# B&R Automation Studio project MotionTestBenchMaster (part 10)

#### Shift_Obj.st
```iecst
FUNCTION_BLOCK PhotoCell_SftObj
	IF IN_ConfigPresent THEN
		VAR_GrippersNumber	:= LIMIT(1, IN_GrippersNumber, CST_RepetitiveArrayDim);
		VAR_Mask 			:= IN_MaskEn AND HMI.Mask;

		IF VAR_Mask THEN
			VAR_Signal := IN_WaitOn AND NOT IN_WaitOff;
		ELSE
			VAR_Signal := IO.DI_Input;
		END_IF

		HMI.On := VAR_Signal;

		OUT	:= HMI.On;

		IF IN_MachinePitch AND IN_Enable THEN
			VAR_ActualValveCounter	:= INT_TO_USINT(FC_ReminderShift(VAR_ActualValveCounter	+ 1, VAR_GrippersNumber, 0));

			IF IN_WritePresenceEnable THEN //v1.63
				SHIFT_Position.ContainerPresence	:= IO.DI_Input;
			END_IF//v1.63

			IF SHIFT_Position.ContainerPresence THEN//v1.63
				IF NOT SHIFT_Position.ContainerBurst	AND	NOT VAR_Mask THEN//v1.63
					IF NOT IO.DI_Input THEN
						HMI.ConsecutiveErrors	:= SEL((IN_MStopConsecutiveValue > 0), 0,HMI.ConsecutiveErrors + 1);
						HMI.AbsoluteErrors		:= SEL((IN_CBlockAbsoluteValue > 0), 0, HMI.AbsoluteErrors + 1);
						HMI.TotalErrors			:= SEL((IN_MStopAbsoluteValue > 0), HMI.TotalErrors, HMI.TotalErrors + 1);

						VAR_RepetitiveCounterArray[VAR_ActualValveCounter]	:= SEL((IN_CBlockRepetitiveValue > 0), 0, VAR_RepetitiveCounterArray[VAR_ActualValveCounter] + 1);
						SHIFT_Position.ContainerPresence	:= FALSE;//v1.63

						IF VAR_RepetitiveCounterArray[VAR_ActualValveCounter] > IN_CBlockRepetitiveValue THEN
							OUT_CBlockRepetitive	:= TRUE;
						END_IF
					ELSE
						VAR_RepetitiveCounterArray[VAR_ActualValveCounter]	:= 0;
						HMI.ConsecutiveErrors	:= 0;//v1.63
					END_IF
				ELSE//v1.63
					VAR_RepetitiveCounterArray[VAR_ActualValveCounter]	:= 0;
					HMI.ConsecutiveErrors	:= 0;
				END_IF//v1.63
			END_IF

			HMI.AlwaysTrueSteps	:= SEL(VAR_EdgeChecked, HMI.AlwaysTrueSteps + 1, 0);//v1.63

			IF IN_CBlockRepetitiveValue > 0 THEN
				HMI.RepetitiveErrors	:= 0;

				FOR VAR_GrippersNumber:= 1	TO	CST_RepetitiveArrayDim	DO
					HMI.RepetitiveErrors := MAX(HMI.RepetitiveErrors, VAR_RepetitiveCounterArray[VAR_GrippersNumber]);
				END_FOR
			END_IF
		ELSIF NOT IO.DI_Input AND IN_Enable THEN
			VAR_EdgeChecked		:= TRUE;
		END_IF

		TMR_TON_TotalCounterReset(IN := IN_ResetCounters OR HMI.CounterReset, PT := T#5s);

		IF IN_ResetCounters OR HMI.CounterReset OR VAR_Mask OR NOT IN_Enable THEN
			IF NOT VAR_CounterResetMemory THEN
				VAR_CounterResetMemory	:= TRUE;

				FOR VAR_GrippersNumber:= 1 TO CST_RepetitiveArrayDim DO
					VAR_RepetitiveCounterArray[VAR_GrippersNumber]	:= 0;
					OUT_CBlockRepetitive	:= FALSE;
				END_FOR

				HMI.AlwaysTrueSteps		:= 0;
				HMI.RepetitiveErrors	:= 0;
				HMI.ConsecutiveErrors	:= 0;
				HMI.AbsoluteErrors		:= 0;
			END_IF
		ELSE
			VAR_CounterResetMemory	:= FALSE;
		END_IF

		IF TMR_TON_TotalCounterReset.Q THEN
			IF NOT VAR_TotalCounterResetMemory THEN
				VAR_TotalCounterResetMemory := TRUE;
				HMI.TotalErrors	:= 0;
			END_IF
		ELSE
			VAR_TotalCounterResetMemory := FALSE;
		END_IF

		HMI.ConfigPresent 	:= IN_ConfigPresent;
		HMI.ConfigAlarm 	:= IN_Alarm;
		HMI.Alarm 			:= OUT_CBlockAbsolute OR OUT_MStopConsecutive OR OUT_MStopAbsolute OR OUT_AlwaysTrueError;
		HMI.Wait			:= (IN_WaitOn AND NOT HMI.On) OR (IN_WaitOff AND HMI.On);
		HMI.MaskEnable		:= IN_MaskEn;

		OUT_CBlockAbsolute		:= (HMI.AbsoluteErrors 		>= IN_CBlockAbsoluteValue)		AND (IN_CBlockAbsoluteValue		> 0);
		OUT_MStopConsecutive	:= (HMI.ConsecutiveErrors 	>= IN_MStopConsecutiveValue)	AND (IN_MStopConsecutiveValue	> 0);
		OUT_MStopAbsolute		:= (HMI.AbsoluteErrors 		>= (IN_MStopAbsoluteValue + IN_CBlockAbsoluteValue))		AND (IN_MStopAbsoluteValue		> 0);	//V4.A.A.1.6.12
		OUT_AlwaysTrueError		:= (HMI.AlwaysTrueSteps		>= CST_AlwaysTrueMaxSteps)		AND (CST_AlwaysTrueMaxSteps		> 0);
	ELSE
		OUT						:= FALSE;
		OUT_CBlockRepetitive	:= FALSE;
		OUT_CBlockAbsolute		:= FALSE;
		OUT_MStopConsecutive	:= FALSE;
		OUT_MStopAbsolute		:= FALSE;
		OUT_AlwaysTrueError		:= FALSE;
		HMI.On 					:= FALSE;
		HMI.MaskEnable			:= FALSE;
		HMI.ConfigPresent 		:= FALSE;
		HMI.ConfigAlarm 		:= FALSE;
		HMI.Alarm 				:= FALSE;
		HMI.Wait				:= FALSE;
		HMI.RepetitiveErrors	:= 0;
		HMI.ConsecutiveErrors	:= 0;
		HMI.AbsoluteErrors		:= 0;
		HMI.AlwaysTrueSteps		:= 0;
	END_IF
END_FUNCTION_BLOCK

FUNCTION_BLOCK CapPhotoCell_SftObj
	IF IN_ConfigPresent THEN
		VAR_GrippersNumber	:= LIMIT(1, IN_GrippersNumber, CST_CounterArrayDim);
		VAR_Mask 			:= IN_MaskEn AND HMI.Mask;

		IF VAR_Mask THEN
			VAR_Signal := IN_WaitOn AND NOT IN_WaitOff;
		ELSE
			VAR_Signal := IO.DI_Input;
		END_IF

		HMI.On := VAR_Signal;

		OUT	:= HMI.On;

		IF IN_MachinePitch AND IN_Enable THEN
			VAR_ActualValveCounter	:= INT_TO_USINT(FC_ReminderShift(VAR_ActualValveCounter + 1, VAR_GrippersNumber, 0));

			IF SHIFT_Position.ContainerPresence AND SHIFT_Position.ClosingReleased AND NOT VAR_Mask THEN
				HMI.AlwaysTrueSteps	:= SEL(VAR_EdgeChecked, HMI.AlwaysTrueSteps + 1, 0);
				SHIFT_Position.ContainerClosed	:= IO.DI_Input;

				IF VAR_CapsReleased < 16#FFFFFFFF THEN
					VAR_CapsReleased := VAR_CapsReleased + 1;
				ELSE
					FOR VAR_i := VAR_AbsoluteErrorN TO 1 BY -1 DO
						VAR_AbsoluteCounterArray[VAR_i] := VAR_AbsoluteCounterArray[VAR_i] - (VAR_AbsoluteCounterArray[1] - 1);
					END_FOR
					VAR_CapsReleased := VAR_AbsoluteCounterArray[VAR_AbsoluteErrorN] + 1;
				END_IF

				IF NOT IO.DI_Input THEN
					HMI.ConsecutiveErrors	:= SEL((IN_MStopConsecutiveValue > 0), 0,HMI.ConsecutiveErrors + 1);
					//HMI.AbsoluteErrors		:= SEL((IN_CBlockAbsoluteValue > 0), 0, VAR_AbsoluteErrorN);	//V4.A.A.1.6.12
					HMI.TotalErrors			:= SEL((IN_CBlockAbsoluteValue > 0) OR (IN_MStopConsecutiveValue > 0), HMI.TotalErrors, HMI.TotalErrors + 1);

					VAR_RepetitiveCounterArray[VAR_ActualValveCounter] := SEL((IN_CBlockRepetitiveValue > 0), 0, VAR_RepetitiveCounterArray[VAR_ActualValveCounter] + 1);

					IF VAR_RepetitiveCounterArray[VAR_ActualValveCounter] > IN_CBlockRepetitiveValue THEN
						OUT_CBlockRepetitive	:= TRUE;
					END_IF

					IF IN_CBlockAbsoluteValue > 0 THEN
						IF IN_CBlockAbsoluteQuantity > 0 THEN
							VAR_AbsoluteCounterArray[VAR_AbsoluteErrorN] := VAR_CapsReleased;
						ELSE
							VAR_AbsoluteCounterArray[VAR_AbsoluteErrorN] := 0;
						END_IF

						VAR_AbsoluteErrorN := VAR_AbsoluteErrorN + 1;
					ELSE
						VAR_AbsoluteCounterArray[VAR_AbsoluteErrorN] := 0;
						VAR_AbsoluteErrorN := 1;
					END_IF
				ELSE
					VAR_RepetitiveCounterArray[VAR_ActualValveCounter]	:= 0;
					HMI.ConsecutiveErrors	:= 0; //v1.7.4
				END_IF
//			ELSE 								//v1.7.4
//				HMI.ConsecutiveErrors	:= 0;	//v1.7.4
			END_IF

			IF ((VAR_CapsReleased - VAR_AbsoluteCounterArray[1]) > IN_CBlockAbsoluteQuantity) AND (IN_CBlockAbsoluteQuantity > 0) THEN
				memmove(ADR(VAR_AbsoluteCounterArray[1]), ADR(VAR_AbsoluteCounterArray[2]), SIZEOF(VAR_AbsoluteCounterArray[1]) * 49);
				VAR_AbsoluteCounterArray[50] := 0;
				VAR_AbsoluteErrorN := MAX(VAR_AbsoluteErrorN - 1, 1);
			END_IF

			IF IN_CBlockRepetitiveValue > 0 THEN
				HMI.RepetitiveErrors := 0;
				FOR VAR_GrippersNumber:= 1 TO CST_CounterArrayDim DO
					HMI.RepetitiveErrors := MAX(HMI.RepetitiveErrors, VAR_RepetitiveCounterArray[VAR_GrippersNumber]);
				END_FOR
			END_IF

			HMI.AbsoluteErrors		:= SEL((IN_CBlockAbsoluteValue > 0), 0, VAR_AbsoluteErrorN - 1);	//V4.A.A.1.6.12
		ELSIF NOT IO.DI_Input AND IN_Enable THEN
			VAR_EdgeChecked := TRUE;
		ELSIF NOT IN_Enable THEN
			SHIFT_Position.ContainerClosed	:= SHIFT_Position.ContainerPresence AND SHIFT_Position.ClosingReleased;
		END_IF

		TMR_TON_TotalCounterReset(IN := IN_ResetCounters OR HMI.CounterReset, PT := T#5s);

		IF IN_ResetCounters OR HMI.CounterReset OR VAR_Mask OR NOT IN_Enable THEN
			IF NOT VAR_CounterResetMemory THEN
				VAR_CounterResetMemory	:= TRUE;

				FOR VAR_GrippersNumber:= 1 TO CST_CounterArrayDim DO
					VAR_RepetitiveCounterArray[VAR_GrippersNumber]	:= 0;
					OUT_CBlockRepetitive	:= FALSE;
				END_FOR

				memset(ADR(VAR_AbsoluteCounterArray[1]), 0, SIZEOF(VAR_AbsoluteCounterArray));
				VAR_AbsoluteErrorN := 1;

				VAR_CapsReleased		:= 0;
				HMI.AlwaysTrueSteps		:= 0;
				HMI.RepetitiveErrors	:= 0;
				//HMI.ConsecutiveErrors	:= 0;//V1.61
				HMI.AbsoluteErrors		:= 0;
			END_IF
		ELSE
			VAR_CounterResetMemory	:= FALSE;
		END_IF
		(*V1.61 Consecutive Errorors counter reset new management*)
		IF IN_ResetCountersConsecutive OR VAR_Mask OR NOT IN_Enable THEN
			IF NOT VAR_CounterConsResetMemory THEN
				VAR_CounterConsResetMemory	:= TRUE;
				HMI.ConsecutiveErrors	:= 0;
			END_IF
		ELSE
			VAR_CounterConsResetMemory	:= FALSE;
		END_IF

		IF TMR_TON_TotalCounterReset.Q THEN
			IF NOT VAR_TotalCounterResetMemory THEN
				VAR_TotalCounterResetMemory := TRUE;
				HMI.TotalErrors	:= 0;
			END_IF
		ELSE
			VAR_TotalCounterResetMemory := FALSE;
		END_IF

		HMI.ConfigPresent 	:= IN_ConfigPresent;
		HMI.ConfigAlarm 	:= IN_Alarm;
		HMI.Alarm 			:= OUT_CBlockAbsolute OR OUT_MStopConsecutive OR OUT_AlwaysTrueError;
		HMI.Wait			:= (IN_WaitOn AND NOT HMI.On) OR (IN_WaitOff AND HMI.On);
		HMI.MaskEnable		:= IN_MaskEn;

		OUT_CBlockAbsolute		:= (HMI.AbsoluteErrors 		>= IN_CBlockAbsoluteValue)		AND (IN_CBlockAbsoluteValue		> 0);
		OUT_MStopConsecutive	:= (HMI.ConsecutiveErrors 	>= IN_MStopConsecutiveValue)	AND (IN_MStopConsecutiveValue	> 0);
		OUT_AlwaysTrueError		:= (HMI.AlwaysTrueSteps		>= CST_AlwaysTrueMaxSteps)		AND (CST_AlwaysTrueMaxSteps		> 0);
	ELSE
		OUT						:= FALSE;
		OUT_CBlockRepetitive	:= FALSE;
		OUT_CBlockAbsolute		:= FALSE;
		OUT_MStopConsecutive	:= FALSE;
		OUT_AlwaysTrueError		:= FALSE;
		HMI.On 					:= FALSE;
		HMI.MaskEnable			:= FALSE;
		HMI.ConfigPresent 		:= FALSE;
		HMI.ConfigAlarm 		:= FALSE;
		HMI.Alarm 				:= FALSE;
		HMI.Wait				:= FALSE;
		HMI.RepetitiveErrors	:= 0;
		HMI.ConsecutiveErrors	:= 0;
		HMI.AbsoluteErrors		:= 0;
		HMI.AlwaysTrueSteps		:= 0;
	END_IF
END_FUNCTION_BLOCK

FUNCTION_BLOCK CapPhotoCell_SftObj_old
	IF IN_ConfigPresent THEN
		VAR_GrippersNumber	:= LIMIT(1, IN_GrippersNumber, CST_RepetitiveArrayDim);
		VAR_Mask 			:= IN_MaskEn AND HMI.Mask;

		IF VAR_Mask THEN
			VAR_Signal := IN_WaitOn AND NOT IN_WaitOff;
		ELSE
			VAR_Signal := IO.DI_Input;
		END_IF

		HMI.On := VAR_Signal;

		OUT	:= HMI.On;

		IF IN_MachinePitch AND IN_Enable THEN
			VAR_ActualValveCounter	:= INT_TO_USINT(FC_ReminderShift(VAR_ActualValveCounter + 1, VAR_GrippersNumber, 0));

			IF SHIFT_Position.ContainerPresence AND SHIFT_Position.ClosingReleased AND NOT VAR_Mask THEN
				HMI.AlwaysTrueSteps	:= SEL(VAR_EdgeChecked, HMI.AlwaysTrueSteps + 1, 0);
				SHIFT_Position.ContainerClosed	:= IO.DI_Input;

				IF NOT IO.DI_Input THEN
					HMI.ConsecutiveErrors	:= SEL((IN_MStopConsecutiveValue > 0), 0,HMI.ConsecutiveErrors + 1);
					HMI.AbsoluteErrors		:= SEL((IN_CBlockAbsoluteValue > 0), 0, HMI.AbsoluteErrors + 1);
					HMI.TotalErrors			:= SEL((IN_MStopAbsoluteValue > 0), HMI.TotalErrors, HMI.TotalErrors + 1);

					VAR_RepetitiveCounterArray[VAR_ActualValveCounter] := SEL((IN_CBlockRepetitiveValue > 0), 0, VAR_RepetitiveCounterArray[VAR_ActualValveCounter] + 1);

					IF VAR_RepetitiveCounterArray[VAR_ActualValveCounter] > IN_CBlockRepetitiveValue THEN
						OUT_CBlockRepetitive	:= TRUE;
					END_IF
				ELSE
					VAR_RepetitiveCounterArray[VAR_ActualValveCounter]	:= 0;
				END_IF
			ELSE
				HMI.ConsecutiveErrors	:= 0;
			END_IF

			IF IN_CBlockRepetitiveValue > 0 THEN
				HMI.RepetitiveErrors := 0;
				FOR VAR_GrippersNumber:= 1 TO CST_RepetitiveArrayDim DO
					HMI.RepetitiveErrors := MAX(HMI.RepetitiveErrors, VAR_RepetitiveCounterArray[VAR_GrippersNumber]);
				END_FOR
			END_IF
		ELSIF NOT IO.DI_Input AND IN_Enable THEN
			VAR_EdgeChecked := TRUE;
		ELSIF NOT IN_Enable THEN
			SHIFT_Position.ContainerClosed	:= SHIFT_Position.ContainerPresence AND SHIFT_Position.ClosingReleased;
		END_IF

		TMR_TON_TotalCounterReset(IN := IN_ResetCounters OR HMI.CounterReset, PT := T#5s);

		IF IN_ResetCounters OR HMI.CounterReset OR VAR_Mask THEN
			IF NOT VAR_CounterResetMemory THEN
				VAR_CounterResetMemory	:= TRUE;

				FOR VAR_GrippersNumber:= 1 TO CST_RepetitiveArrayDim DO
					VAR_RepetitiveCounterArray[VAR_GrippersNumber]	:= 0;
					OUT_CBlockRepetitive	:= FALSE;
				END_FOR

				HMI.AlwaysTrueSteps		:= 0;
				HMI.RepetitiveErrors	:= 0;
				HMI.ConsecutiveErrors	:= 0;
				HMI.AbsoluteErrors		:= 0;
			END_IF
		ELSE
			VAR_CounterResetMemory	:= FALSE;
		END_IF

		IF TMR_TON_TotalCounterReset.Q THEN
			IF NOT VAR_TotalCounterResetMemory THEN
				VAR_TotalCounterResetMemory := TRUE;
				HMI.TotalErrors	:= 0;
			END_IF
		ELSE
			VAR_TotalCounterResetMemory := FALSE;
		END_IF

		HMI.ConfigPresent 	:= IN_ConfigPresent;
		HMI.ConfigAlarm 	:= IN_Alarm;
		HMI.Alarm 			:= OUT_CBlockAbsolute OR OUT_MStopConsecutive OR OUT_MStopAbsolute OR OUT_AlwaysTrueError;
		HMI.Wait			:= (IN_WaitOn AND NOT HMI.On) OR (IN_WaitOff AND HMI.On);
		HMI.MaskEnable		:= IN_MaskEn;

		OUT_CBlockAbsolute		:= (HMI.AbsoluteErrors 		>= IN_CBlockAbsoluteValue)		AND (IN_CBlockAbsoluteValue		> 0);
		OUT_MStopConsecutive	:= (HMI.ConsecutiveErrors 	>= IN_MStopConsecutiveValue)	AND (IN_MStopConsecutiveValue	> 0);
		OUT_MStopAbsolute		:= (HMI.AbsoluteErrors 		>= IN_MStopAbsoluteValue)		AND (IN_MStopAbsoluteValue		> 0);
		OUT_AlwaysTrueError		:= (HMI.AlwaysTrueSteps		>= CST_AlwaysTrueMaxSteps)		AND (CST_AlwaysTrueMaxSteps		> 0);
	ELSE
		OUT						:= FALSE;
		OUT_CBlockRepetitive	:= FALSE;
		OUT_CBlockAbsolute		:= FALSE;
		OUT_MStopConsecutive	:= FALSE;
		OUT_MStopAbsolute		:= FALSE;
		OUT_AlwaysTrueError		:= FALSE;
		HMI.On 					:= FALSE;
		HMI.MaskEnable			:= FALSE;
		HMI.ConfigPresent 		:= FALSE;
		HMI.ConfigAlarm 		:= FALSE;
		HMI.Alarm 				:= FALSE;
		HMI.Wait				:= FALSE;
		HMI.RepetitiveErrors	:= 0;
		HMI.ConsecutiveErrors	:= 0;
		HMI.AbsoluteErrors		:= 0;
		HMI.AlwaysTrueSteps		:= 0;
	END_IF
END_FUNCTION_BLOCK

FUNCTION_BLOCK Ejector_SftObj
	VAR_Mask	:= HMI.Mask AND IN_MaskEn;

	(* Local *)
	IF IN_ManEn AND NOT IN_HMIAutoForce THEN
		VAR_ManOn	:= HMI.ManOn;
		VAR_Auto	:= NOT HMI.ManOff AND NOT HMI.ManOn;
	ELSE
		VAR_ManOn	:= FALSE;
		VAR_Auto	:= TRUE;
		HMI.ManOn	:= FALSE;
		HMI.ManOff	:= FALSE;
	END_IF

	IF IN_MachinePitch THEN
		VAR_AutoCnd := IN_ShiftPosition.ContainerPresence		AND (IN_ShiftPosition.ContainerBurst	OR
						(NOT IN_ShiftPosition.ContainerFilled	AND IN_FillingErrorEject) OR IN_ShiftPosition.EjectContainer) AND NOT VAR_Mask; (*V1.61*)
		IF VAR_AutoCnd AND NOT IN_SamplingModeActive THEN (*V1.61*)
			HMI.ConsecutiveErrors	:= HMI.ConsecutiveErrors	+ 1;
			HMI.AbsoluteErrors		:= HMI.AbsoluteErrors		+ 1;
			HMI.TotalErrors			:= HMI.TotalErrors			+ 1;
		ELSE
			HMI.ConsecutiveErrors	:= 0;
		END_IF(*V1.61*)

		IF IN_SamplingModeActive AND VAR_AutoCnd THEN (*V1.61*)
			IN_ShiftPosition.ContainerEjected := TRUE;(*V1.61*)
		ELSE
			IN_ShiftPosition.ContainerEjected := FALSE;(*V1.61*)
		END_IF
	END_IF

	TMR_TON_TotalCounterReset(IN := IN_ResetCounters OR HMI.CounterReset, PT := T#5s);

	IF IN_ResetCounters OR HMI.CounterReset THEN
		IF NOT VAR_CounterResetMemory THEN
			VAR_CounterResetMemory	:= TRUE;
			HMI.ConsecutiveErrors	:= 0;
			HMI.AbsoluteErrors		:= 0;
		END_IF
	ELSE
		VAR_CounterResetMemory	:= FALSE;
	END_IF

	IF TMR_TON_TotalCounterReset.Q THEN
		IF NOT VAR_TotalCounterResetMemory THEN
			VAR_TotalCounterResetMemory := TRUE;
			HMI.TotalErrors	:= 0;
		END_IF
	ELSE
		VAR_TotalCounterResetMemory := FALSE;
	END_IF

	IF IN_ConfigPresent THEN
		IF IN_Enable THEN
			IF VAR_Auto THEN
				VAR_ValveOpened := VAR_AutoCnd;
			ELSIF VAR_ManOn THEN
				VAR_ValveOpened := TRUE;
			ELSE
				VAR_ValveOpened := FALSE;
			END_IF
		ELSIF NOT IN_ConfigType THEN
			VAR_ValveOpened := FALSE;
		END_IF
		VAR_ValveClosed := NOT VAR_ValveOpened;

		OUT						:= VAR_ValveOpened;
		OUT_CBlockAbsolute		:= (HMI.AbsoluteErrors 		>= IN_CBlockAbsoluteValue)		AND (IN_CBlockAbsoluteValue		> 0);
		OUT_MStopConsecutive	:= (HMI.ConsecutiveErrors 	>= IN_MStopConsecutiveValue)	AND (IN_MStopConsecutiveValue	> 0);
	ELSE
		VAR_ValveOpened			:= FALSE;
		VAR_ValveClosed			:= FALSE;
		OUT						:= FALSE;
		OUT_CBlockAbsolute		:= 0;
		OUT_MStopConsecutive	:= 0;
	END_IF

	(* HMI *)
	HMI.ManEnable		:= IN_ManEn;
	HMI.ConfigPresent	:= IN_ConfigPresent;
	HMI.MaskEnable		:= IN_MaskEn;
	HMI.Alarm 			:= OUT_CBlockAbsolute OR OUT_MStopConsecutive;

	(* IO *)
	IO.DO_Opened	:= VAR_ValveOpened;
	IO.DO_Closed	:= VAR_ValveClosed;
	HMI.Out			:= IO.DO_Opened;
END_FUNCTION_BLOCK
```

#### Constant.var - Global variables
```iecst
VAR CONSTANT
	CST_Valve_Dig_Mono_CFG : USINT := 0;
	CST_Valve_Dig_Bi_CFG : USINT := 1;
	CST_AI_Compare_OFF : USINT := 0; (*FALSE*)
	CST_AI_Compare_LT : USINT := 1; (*PV < SP*)
	CST_AI_Compare_GT : USINT := 2; (*PV > SP*)
	CST_AI_Compare_EQ : USINT := 3; (*PV = SP*)
	CST_AI_Compare_ON : USINT := 4; (*TRUE*)
	CST_AI_FaultMode_Hold : USINT := 0; (*Hold on fault*)
	CST_AI_FaultMode_Low : USINT := 1; (*Low on fault*)
	CST_AI_FaultMode_High : USINT := 2; (*High on fault*)
END_VAR
(*Communication Type*)
VAR CONSTANT
	CST_CFG_NotPresent : USINT := 0;
	CST_CFG_TCP : USINT := 1; (*TCP IP*)
	CST_CFG_ETH : USINT := 2; (*ETHERNET IP*)
	CST_CFG_MODBUS : USINT := 3;
	CST_CFG_PROFIBUS : USINT := 4;
	CST_CFG_POWERLINK : USINT := 5;
	CST_CFG_HW : USINT := 6;
	CST_CFG_UDP : USINT := 7;
	CST_CFG_SCC : USINT := 8;
	CST_CFG_PROFINET : USINT := 9;
	CST_CFG_OPC : USINT := 10;
END_VAR
(*Comparison Constants*)
VAR CONSTANT
	CST_EQ : USINT := 0; (*The equality operator symbol '=' *)
	CST_GE : USINT := 1; (*The greater than or equal to symbol '>=' *)
	CST_LE : USINT := 2; (*The less than or equal to symbol '<='*)
	CST_GT : USINT := 3; (*The greater than operator symbol '>'*)
	CST_LT : USINT := 4; (*The division operator symbol '<'*)
	CST_NE : USINT := 5; (*The unequality operator symbol '<>'*)
END_VAR
```

#### UVtronic_Std.st - not listed in the package file held
```iecst
FUNCTION_BLOCK UVtronic_Std
	IF NOT VAR_FirstCycle THEN
		HMI.ManOff		:= FALSE;
		HMI.ManOn		:= FALSE;
		VAR_FirstCycle	:= TRUE;
	END_IF

	IF IN_ConfigPresent THEN
		(*****************************************************************)
		(*****************************START*******************************)
		(*****************************************************************)
		IF (EDGENEG(IN_ManEn) AND HMI.ManOn) OR IN_HMIAutoForce THEN
			HMI.ManOn	:= FALSE;
			HMI.ManOff	:= FALSE;
		END_IF

		VAR_Mask := HMI.Mask AND IN_MaskEn;
		VAR_Auto := NOT HMI.ManOff AND NOT HMI.ManOn;

		IF VAR_Fault OR NOT IN_Enable THEN
			IO.DO_MotorON := FALSE;
		ELSIF VAR_Auto THEN
			IO.DO_MotorON := IN_AutoCnd;
		ELSE
			IO.DO_MotorON := HMI.ManOn;
		END_IF

		(*****************************************************************)
		(**************************ALARM LOGIC****************************)
		(*****************************************************************)
		TMR_TON(IN := IO.DO_MotorON,
				PT := IN_FBKDelay);

		TMR_TOF(IN := NOT IO.DO_MotorON,
				PT := IN_FBKDelay);

		IF IN_Reset THEN
			VAR_ContactorFBK	:= FALSE;
			VAR_GeneralFault	:= FALSE;
			VAR_Overload		:= FALSE;
			VAR_NotReady		:= FALSE;
		END_IF

		IF ((TMR_TON.Q AND IO.DI_ContactorFBK) OR (TMR_TOF.Q AND NOT IO.DI_ContactorFBK)) AND NOT IN_ConfigType AND NOT VAR_Mask THEN
			VAR_ContactorFBK := NOT IN_Simulation;
		END_IF

		IF IO.DI_GeneralFault AND NOT VAR_Mask THEN
			VAR_GeneralFault := NOT IN_Simulation;
		END_IF

		IF NOT IO.DI_OverloadOK AND NOT IN_ConfigType AND NOT VAR_Mask THEN
			VAR_Overload := NOT IN_Simulation;
		END_IF

		IF NOT IO.DI_Ready AND NOT VAR_Mask THEN
			VAR_NotReady := NOT IN_Simulation;
		END_IF

		VAR_Fault := (VAR_ContactorFBK OR VAR_GeneralFault OR VAR_Overload OR VAR_NotReady AND IN_Enable) AND NOT IN_Simulation;

		(*****************************************************************)
		(******************************HMI********************************)
		(*****************************************************************)
		HMI.Out				:= IO.DO_MotorON;
		HMI.Alarm			:= VAR_Fault;
		HMI.Isolated		:= FALSE;
		HMI.Overload		:= VAR_Overload;
		HMI.FeedBack		:= VAR_ContactorFBK;
		HMI.ConfigPresent	:= IN_ConfigPresent;
		HMI.ManEnable		:= IN_ManEn;
		HMI.MaskEnable		:= IN_MaskEn;

		(*****************************************************************)
		(******************************OUT********************************)
		(*****************************************************************)
		OUT_Running				:= IO.DO_MotorON;
		OUT_NotReady			:= VAR_NotReady;
		OUT_GeneralFault		:= VAR_GeneralFault;
		OUT_ContactorFBKFault	:= VAR_ContactorFBK;
		OUT_OverloadFault		:= VAR_Overload;
		OUT_Alarm				:= VAR_Fault;
	ELSE
		memset(ADR(HMI), 0, SIZEOF(HMI));
		OUT_Running				:= FALSE;
		OUT_NotReady			:= FALSE;
		OUT_GeneralFault		:= FALSE;
		OUT_ContactorFBKFault	:= FALSE;
		OUT_OverloadFault		:= FALSE;
		OUT_Alarm				:= FALSE;
		IO.DO_MotorON			:= FALSE;
	END_IF
END_FUNCTION_BLOCK
```

### Library Logical/00_AID/Libraries/Sidel_Libraries/ITC/MBTCP (ANSIC, version 0.01.0) - ModBusTCP
Depends on: Runtime, standard, AsTCP, sys_lib, brsystem, asstring

#### MBTCP.fun - Exported functions and function blocks
```iecst
(********************************************************************
 * COPYRIGHT -- Bernecker + Rainer
 ********************************************************************
 * Library: MBTCP
 * File: MBTCP.fun
 * Author: B&R
 * Created: September 04, 2008
 ********************************************************************
 * Functions and function blocks of library MBTCP
 ********************************************************************)
(*Configures a Modbus over TCP slave (server) and provides a Modbus slave ID. fMBTSOpen() should be called in the INIT section of a task prior to fMBTSlave(). See also fMBTSClose() to close the slave in the EXIT section. This slave can then be read from, or written to, by fMBTMaster() or widely available Modbus over TCP programs.Hosts up to 127 Modbus units, each unit contains set of size-adjustable coils, discrete inputs, input registers, and holding registers. <a href="../MBTCP_Server.html"> See Modbus Slave/Server for more information</a>*)

FUNCTION_BLOCK fMBTSOpen
	VAR_INPUT
		bEnable : BOOL; (*Enables the function block*)
		uiPort : UINT; (*TCP port number (default = 502) *)
		uiNbrCoils : UINT; (*Number of read-write binary coils*)
		uiNbrDiscreteInputs : UINT; (*Number of read-only binary discrete inputs *)
		uiNbrInputRegs : UINT; (*Number of read-only 16-bit input registers *)
		uiNbrHoldingRegs : UINT; (*Number of read-write 16-bit holding registers *)
		uiOffsetUnits : UINT; (*Offset of Modbus units. *)
		uiNbrUnits : UINT; (*Number of Modbus units. If external array are used this parameter has to be set to 1*)
		pbCoil : REFERENCE TO BOOL; (*Coil mapping, given as array of BOOL. Must be set to 0 if internal mapping is used*)
		pbDInp : REFERENCE TO BOOL; (*Discrete input mapping, given as array of BOOL. Must be set to 0 if internal mapping is used*)
		puiIReg : REFERENCE TO UINT; (*Input register mapping, given as array of UINT. Must be set to 0 if internal mapping is used*)
		puiHReg : REFERENCE TO UINT; (*Holding register mapping, given as array of UINT. Must be set to 0 if internal mapping is used*)
	END_VAR
	VAR_OUTPUT
		uiNbrAllocUnits : UINT; (*Number of actaully allocated units *)
		udiIdent : UDINT; (*Ident (pointer to memory area holding Modbus server structure)*)
		uiStatus : UINT; (*Status 0 for OK, otherwise <a href="../../Data_types_and_constants/Constants.html"> Error Number </a>*)
	END_VAR
END_FUNCTION_BLOCK
(*Modbus/TCP slave (server) function. fMBTSlave() should be called in the CYCLIC section of a task after being configured by fMBTSOpen(). The server is closed by fMBTSClose(). This server can be read from or written to by fMBTMaster() or widely available Modbus over TCP programs. <a href="../MBTCP_Server.html"> See Modbus Slave/Server for more information</a>*)

FUNCTION_BLOCK fMBTSlave
	VAR_INPUT
		bEnable : BOOL; (*Enables the function block*)
		udiIdent : UDINT; (*Ident, as provided in instfMBTSOpen.udiIdent *)
		tiRecvDelay : TIME; (*Time to wait before disconnecting a non-responding client (master)*)
	END_VAR
	VAR_OUTPUT
		usiClientNbr : UINT; (*How many clients (masters) are connected *)
		usiClientServed : USINT; (*Client (master) currently served *)
		tiRecvElapsed : TIME; (*Time spent waiting for response from Master *)
		usiUnit : USINT; (*Server unit read or written *)
		usiClientIP : STRING[18]; (*Client (master) IP address *)
		usiMBFuncCode : USINT; (*Modbus function code *)
		uiSentDataLen : UINT; (*Length of data sent *)
		szMsg : STRING[100]; (*Debug Message*)
		stTcpServerStatus : UINT; (*Status from the TCPServer function*)
		udiRecvCnt : UDINT; (*Counter receive data*)
		udiSendCnt : UDINT; (*Counter Send Data*)
		usiOpenRetries : USINT; (*Port open Retries*)
		CltInfo : ARRAY[0..4] OF tstclient_info; (*Client Info (IP-Adresse, Port, Ident)*)
		uiStep : UINT; (*Current step executed by the Slave's state machine*)
		uiStatus : UINT; (*Status 0 for OK, otherwise <a href="../../Data_types_and_constants/Constants.html"> Error Number </a>*)
	END_VAR
END_FUNCTION_BLOCK
(*Terminates a Modbus/TCP slave (server) and releases allocated memory. fMBTSClose() should be called in the EXIT section of a task. See also fMBTSOpen() and fMBTSlave().*)

FUNCTION_BLOCK fMBTSClose
	VAR_INPUT
		bEnable : BOOL; (*Enables the function block*)
		udiIdent : UDINT; (*Ident, as provided in instfMBTSOpen.udiIdent *)
	END_VAR
	VAR_OUTPUT
		uiStatus : UINT; (*Status 0 for OK, otherwise <a href="../../Data_types_and_constants/Constants.html"> Error Number </a>*)
	END_VAR
END_FUNCTION_BLOCK
(*Read/write individual values from/to coils and registers of given unit. The function code to use in member uiFcode of the passed structure is the same as for Modbus (0x01..0x06,0x0F,0x10,0x17) and two user defined functions (0x41,0x42). *)

FUNCTION_BLOCK fMBTSRW
	VAR_INPUT
		bEnable : BOOL; (*Enables the function block*)
		udiIdent : UDINT; (*Ident, as provided in instfMBTSOpen.udiIdent *)
		usiFCode : USINT; (*Modbus function code, see <a href="../../Data_types_and_constants/Constants.html">constants</a>*)
		usiUnit : USINT; (*Unit to access*)
		uiReadAddr : UINT; (*Element in coil or register for read access*)
		uiReadQty : UINT; (*Quantity of coils/regs to read*)
		puiReadVal : REFERENCE TO UINT; (*Requested read value, pointer to UINT*)
		uiWriteAddr : UINT; (*Element in coil or register for write access*)
		uiWriteQty : UINT; (*Quantity of coils/regs to write*)
		puiWriteVal : REFERENCE TO UINT; (*Requested write value, pointer to UINT*)
	END_VAR
	VAR_OUTPUT
		uiStatus : UINT; (*Status 0 for OK, otherwise <a href="../../Data_types_and_constants/Constants.html"> Error Number </a>*)
	END_VAR
END_FUNCTION_BLOCK
(*Initialize the slave's data units (coils and registers) with values. Coils and Discrete Inputs are initialized with 0, 1, 0... Input registers are filled with 1000, 1001, 1002... Holding registers are initialized with 0, 1, 2... *)

FUNCTION_BLOCK fMBTSFill
	VAR_INPUT
		bEnable : BOOL; (*Enables the function block*)
		udiIdent : UDINT; (*Ident, as provided in instfMBTSOpen.udiIdent *)
	END_VAR
	VAR_OUTPUT
		uiStatus : UINT; (*Status 0 for OK, otherwise <a href="../../Data_types_and_constants/Constants.html"> Error Number </a>*)
	END_VAR
END_FUNCTION_BLOCK
(*Allocates memory and pre-configures Modbus TCP Master. fMBTMOpen() should be called in the INIT section of a task prior to fMBTMaster(). See also fMBTMClose() to close the master in the task's EXIT section. The master connects to the Modbus TCP slave available at the IP address provided by szSlvIPAddr. *)

FUNCTION_BLOCK fMBTMOpen
	VAR_INPUT
		bEnable : BOOL; (*Enables the function block*)
		szSlvIPAddr : STRING[18]; (*Slave's IP address *)
		uiPort : UINT; (*TCP port number (default = 502) *)
		uiRecvTimeout : UINT; (*Timeout to wait for answer from Slave prior to sending new request (default = 500 s) *)
	END_VAR
	VAR_OUTPUT
		udiIdent : UDINT; (*Ident (pointer to memory area holding Modbus Master structure)*)
		uiStatus : UINT; (*Status 0 for OK, otherwise <a href="../../Data_types_and_constants/Constants.html"> Error Number </a>*)
	END_VAR
END_FUNCTION_BLOCK
(*Modbus/TCP master (client) function. fMBTMaster() should be called in the CYCLIC section of a task after being configured by fMBTMOpen(). The master is closed by fMBTMClose(). This master writes to or reads from a slave running fMBTSlave() or other widely available Modbus over TCP slave programs. *)

FUNCTION_BLOCK fMBTMaster
	VAR_INPUT
		bEnable : BOOL; (*Enables the function block*)
		udiIdent : UDINT; (*Ident, as provided in instfMBTMOpen.udiIdent *)
	END_VAR
	VAR_OUTPUT
		uiStep : UINT; (*Step executed by Master. Useful to monitor execution. *)
		uiTxID : UINT; (*Transaction ID *)
		usiMBFuncCode : USINT; (*Modbus function code *)
		szMsg : STRING[100]; (*Status from the TCPClient functions*)
		usiRxByteCnt : USINT; (*Number of bytes received from slave. See response byte count in Modbus protocol. *)
		uiStatus : UINT; (*Status 0 for OK, otherwise <a href="../../Data_types_and_constants/Constants.html"> Error Number </a>*)
	END_VAR
END_FUNCTION_BLOCK
(*Terminates a Modbus/TCP master (client) and releases allocated memory. fMBTMClose() should be called in the EXIT section of a task. See also fMBTMOpen() and fMBTMaster(). *)

FUNCTION_BLOCK fMBTMClose
	VAR_INPUT
		bEnable : BOOL; (*Enables the function block*)
		udiIdent : UDINT; (*Ident, as provided in instfMBTMOpen.udiIdent *)
	END_VAR
	VAR_OUTPUT
		uiStatus : UINT; (*Status 0 for OK, otherwise <a href="../../Data_types_and_constants/Constants.html"> Error Number </a>*)
	END_VAR
END_FUNCTION_BLOCK
(*Read/write individual values from/to coils and registers of given unit. The function code to use in member uiFcode of the passed structure is the same as for Modbus (0x01..0x06,0x0F,0x10,0x17).*)

FUNCTION_BLOCK fMBTMRW
	VAR_INPUT
		bEnable : BOOL; (*Enables the function block*)
		udiIdent : UDINT; (*Ident from fMBTMOpen*)
		usiFCode : USINT; (*Modbus function code, see <a href="../../Data_types_and_constants/Constants.html">constants</a>*)
		usiUnit : USINT; (*Slave unit*)
		uiReadAddr : UINT; (*Element in coil or register for read access*)
		uiReadQty : UINT; (*Quantity of coils/regs to read*)
		puiReadVal : REFERENCE TO UINT; (*Requested read value, pointer to UINT*)
		uiWriteAddr : UINT; (*Element in coil or register for write access*)
		uiWriteQty : UINT; (*Quantity of coils/regs to write*)
		puiWriteVal : REFERENCE TO UINT; (*Requested write value, pointer to UINT*)
		bPoll : BOOL; (*Poll slave repeatedly (0 = single request)*)
		udiPollPeriod : UDINT; (*Polling period in ms*)
	END_VAR
	VAR_OUTPUT
		bRecvOK : BOOL; (*Confirms requested data was sent by slave*)
		uiStatus : UINT; (*Status 0 for OK, otherwise <a href="../../Data_types_and_constants/Constants.html"> Error Number </a>*)
	END_VAR
END_FUNCTION_BLOCK
```

#### MBTCP.typ - Exported data types
```iecst
(********************************************************************
 * COPYRIGHT -- Bernecker + Rainer
 ********************************************************************
 * Library: MBTCP
 * File: MBTCP.typ
 * Author: B&R
 * Created: September 04, 2008
 ********************************************************************
 * Data types of library MBTCP
 ********************************************************************)
(*Client informationen*)

TYPE
	tstclient_info : 	STRUCT  (*Client information*)
		udiIdent : UDINT; (*Client Indentifier*)
		usiPort : USINT; (*Client Port*)
		szIp_addr : STRING[18]; (*Client IP- Adresse*)
		szMsg : STRING[100]; (*Client Message*)
	END_STRUCT;
END_TYPE
```

#### MBTCP.var - Exported constants
```iecst
(********************************************************************
 * COPYRIGHT -- Bernecker + Rainer
 ********************************************************************
 * Library: MBTCP
 * File: MBTCP.var
 * Author: B&R
 * Created: September 04, 2008
 ********************************************************************
 * Constants of library MBTCP <header> Error numbers below 50000 are from automation studio libraries and these are described in the automation studio help. </header>
 ********************************************************************)
VAR CONSTANT
	mbtERR_ILLEGAL_FUNCTION : UINT := 50001; (*Modbus function not implemented/non-existent *)
	mbtERR_DATA_ADDRESS : UINT := 50002; (*Address not available in coil or register *)
	mbtERR_IP_ADRESS : UINT := 50004; (*Wrong IP address passed to Master *)
	mbtERR_NBR_UNITS : UINT := 50005; (*Requested unit does not exist *)
	mbtERR_NULL_POINTER : UINT := 50006; (*Null pointer passed to function block *)
	mbtERR_MAX_CLIENT : UINT := 51001; (*Maximal amount of client is already connected *)
	mbtERR_NOT_CONNECTED : UINT := 51002; (*Half-open connection*)
	mbtERR_WR_ERROR_SOCKET : UINT := 51003; (*TCPServer socket error *)
	mbtERR_FATAL_ERROR : UINT := 51004; (*Fatal Error*)
	mbtERR_TIMEOUT : UINT := 51005; (*Modbus TCP timeout *)
	mbtERR_OPEN_RETRIES_IOC : UINT := 51006; (*Retried open port at the TCP IOControl *)
	mbtERR_OPEN_RETRIES_WR : UINT := 51007; (*Retried open port again at the TCPServer *)
	mbtERR_REQUEST_LEN_ZERO : UINT := 51008; (*The Server received a request with zero bytes *)
	mbtERR_MIN_FRAME_LEN : UINT := 51009; (*The Server received a request with a too short frame*)
	mbtERR_REQUEST_UNIT : UINT := 51010; (*Unit ID too high or low*)
	mbtERR_PROTOCOL_ID : UINT := 51011; (*Protocol ID != 0. Modbus Protocol ID must be 0 *)
	mbtERR_FCODE_ZERO : UINT := 51012; (*Function code is zero*)
	mbtERR_REQUEST : UINT := 51013; (*Request from client is wrong *)
	mbtERR_RESPONSE : UINT := 51014; (*Response from server is wrong *)
	mbtERR_MAX_NBR_COILS : UINT := 51015; (*Maximal number of coils is exceeded (2000) *)
	mbtERR_MAX_NBR_REGISTER : UINT := 51016; (*Maximal number of register is exceeded (127) *)
	mbtEVENT_OPEN_PORT : UINT := 52001; (*Opened new TCP Port *)
	mbtEVENT_ADD_CLIENT : UINT := 52002; (*Added new Client to the MBTCP Server*)
	mbtEVENT_IPADRESS_IDENT : UINT := 52003; (*Deploy ID with IP-adress. The ID is written in binary data at the logger*)
	mbtEVENT_CLOSE_CLIENT : UINT := 52004; (*Closed the Client connection *)
	mbtEVENT_CLOSE_PORT : UINT := 52005; (*Closed the Port*)
	MBT_READ_COILS : USINT := 1; (*Modbus function code: Read coils*)
	MBT_READ_DISCRETE_INPUTS : USINT := 2; (*Modbus function code: Read discrete inputs*)
	MBT_READ_HOLDING_REGISTERS : USINT := 3; (*Modbus function code: Read holding registers*)
	MBT_READ_INPUT_REGISTERS : USINT := 4; (*Modbus function code: Read input registers*)
	MBT_WRITE_SINGLE_COIL : USINT := 5; (*Modbus function code: Write single coil*)
	MBT_WRITE_SINGLE_REGISTER : USINT := 6; (*Modbus function code: Write single register (holding register)*)
	MBT_WRITE_MULTIPLE_COILS : USINT := 15; (*Modbus function code: Write multiple coils*)
	MBT_WRITE_MULTIPLE_REGISTERS : USINT := 16; (*Modbus function code: Write multiple registers (holding register)*)
	MBT_READ_WRITE_MULTIPLE_REGISTER : USINT := 23; (*Modbus function code: Read and write multiple registers*)
	BR_MBT_WRITE_DISCRETE_INPUTS : USINT := 65; (*User defined modbus function code: Write discrete inputs*)
	BR_MBT_WRITE_INPUT_REGISTERS : USINT := 66; (*User defined modbus function code: Write input register*)
END_VAR
```

#### fMBTSOpen.c
```c
/******************************************************************************
 * Copyright:    B&R Industrie-Automation AG
 *
 * Project:      Library MBTCP
 *
 * Target:       B&R-PCC
 *
 * AR-Version:   B 2.01
 *
 * AS-Version:   V 3.0.71.16.SP01
 *
 * Filename:     fMBTSOpen.c
 *
 * Function:     module-description
 *
 * Dependencies: description of all dependencies
 *
 ******************************************************************************
 * History:
 *
 * Version | Date        | Author       | Description
 * ----------------------------------------------------------------------------
 *    1.00 | 2008-sep-19 | H.Anderes    | creation
 *****************************************************************************/

/*****************************************************************************
 * includes
 *****************************************************************************/
/* ansi-c import */
/* system import */
/* user defined import */
#include "MBTCP.h"
#include "MBTSlave.h"

/*****************************************************************************
 * type definitions
 *****************************************************************************/

/*****************************************************************************
 * functions
 *****************************************************************************/
/*===========================================================================*/
void fMBTSOpen(struct fMBTSOpen* inst)
/*----------------------------------------------------------------------------
  Function:

  Configures a Modbus over TCP slave (server) and provides a Modbus
  slave ID. fMBTSOpen() should be called in the INIT section of a task
  prior to fMBTSlave(). See also fMBTSClose() to close the slave in
  the EXIT section. This slave can then be read from, or written to,
  by fMBTMaster() or widely available Modbus over TCP programs.

  History:

  Version | Date        | Author      | Description
  ----------------------------------------------------------------------------
  1.00    | 2008-sep-19 | H.Anderes   | creation
  1.01    | 2009-dez-03 | H.Anderes   | external structures
  ===========================================================================*/
{
  /* _LOCAL */
  UINT astatus    = 0;
  UINT i, u       = 0;
  BOOL extMapping = 0;
  /* _DYNAMIC */
  tstMBT_SVars *mbs;
  tstMBT_SData *pData;
  tCOIL *pCoils;
  tDINP *pDiscreteInputs;
  tIREG *pInputRegs;
  tHREG *pHoldingRegs;
  /*=========================================================================*/
  if (inst == NULL)
  {
    inst->uiStatus = mbtERR_NULL_POINTER;
    goto END;
  }
  if (inst->bEnable < TRUE)
  {
    inst->uiNbrAllocUnits = 0;
    inst->uiStatus = ERR_FUB_ENABLE_FALSE;
  }
  else
  {
    inst->uiStatus = ERR_FUB_BUSY;
    if (inst->uiPort < 1)
      inst->uiPort = MBT_SLAVE_PORT;

    if (inst->uiNbrUnits < 1)
      inst->uiNbrUnits = NUNITS_DEF;

   	if(inst->uiOffsetUnits > 255)
   	 { inst->uiStatus = mbtERR_NBR_UNITS; goto END; }

   	if((inst->uiOffsetUnits + inst->uiNbrUnits) > 256)
   	 { inst->uiStatus = mbtERR_NBR_UNITS; goto END; }

    astatus = TMP_alloc(sizeof(tstMBT_SVars), (void**)&mbs);
    if (astatus > 0) { inst->uiStatus = astatus; goto END; }
    memset(mbs, 0, sizeof(tstMBT_SVars));
    astatus = TMP_alloc(sizeof(tstMBT_SData), (void**)&pData);
    if (astatus > 0) { inst->uiStatus = astatus; goto END; }
    memset(pData, 0, sizeof(tstMBT_SData));
    mbs->pData = pData;

    /* allocate memory for coils and registers
     */
    mbs->pData->uiNbrUnits 		 = inst->uiNbrUnits;
    mbs->pData->uiOffsetUnits = inst->uiOffsetUnits;

    inst->uiNbrAllocUnits = 0;           /* num of allocated units */

   /* check if the mapping type is valid */
   if (   (inst->pbCoil  == NULL)
       && (inst->pbDInp  == NULL)
       && (inst->puiIReg == NULL)
       && (inst->puiHReg == NULL))
   {
     extMapping = FALSE;
   }
   else
   {
     extMapping = TRUE;
   }

    for (u = inst->uiOffsetUnits; u < (inst->uiNbrUnits + inst->uiOffsetUnits); u++)
    {
      if (    (inst->pbCoil == NULL)
           && (inst->uiNbrCoils > 0))
      {
        astatus = TMP_alloc(inst->uiNbrCoils * sizeof(tCOIL),
                            (void **) &pCoils);
        if (astatus > 0) { inst->uiStatus = astatus; goto END; }
        memset((tCOIL *) pCoils, 0,
               inst->uiNbrCoils * sizeof(tCOIL));
        mbs->pData->stUnit[u].pCoils = (tCOIL *) pCoils;
        mbs->pData->stUnit[u].uiNbrCoils = inst->uiNbrCoils;
      }
      else if (    (inst->pbCoil != NULL)
                && (inst->uiNbrCoils > 0))
      {
        mbs->pData->stUnit[u].pCoils       = (tCOIL *) inst->pbCoil;
        mbs->pData->stUnit[u].uiNbrCoils   = inst->uiNbrCoils;
        mbs->pData->stUnit[0].bCoilsExtern = TRUE;
      }

      if (    (inst->pbDInp == NULL)
           && (inst->uiNbrDiscreteInputs > 0))
      {
        astatus = TMP_alloc(inst->uiNbrDiscreteInputs * sizeof(tDINP),
                            (void **) &pDiscreteInputs);
        if (astatus > 0) { inst->uiStatus = astatus; goto END; }
        memset((tDINP *) pDiscreteInputs, 0,
               inst->uiNbrDiscreteInputs * sizeof(tDINP));
        mbs->pData->stUnit[u].pDiscreteInputs = (tDINP *) pDiscreteInputs;
        mbs->pData->stUnit[u].uiNbrDiscreteInputs = inst->uiNbrDiscreteInputs;
      }
      else
      {
        mbs->pData->stUnit[u].pDiscreteInputs        = (tDINP *)  inst->pbDInp;
        mbs->pData->stUnit[u].uiNbrDiscreteInputs    = inst->uiNbrDiscreteInputs;
        mbs->pData->stUnit[0].bDiscreteInputsExtern  = TRUE;
      }

      if (    (inst->puiIReg == NULL)
           && (inst->uiNbrInputRegs > 0))
      {
        astatus = TMP_alloc(inst->uiNbrInputRegs * sizeof(tIREG),
                            (void **) &pInputRegs);
        if (astatus > 0) { inst->uiStatus = astatus; goto END; }
        memset((tIREG *) pInputRegs, 0,
               inst->uiNbrInputRegs * sizeof(tIREG));
        mbs->pData->stUnit[u].pInputRegs = (tIREG *) pInputRegs;
        mbs->pData->stUnit[u].uiNbrInputRegs = inst->uiNbrInputRegs;
      }
      else
      {
        mbs->pData->stUnit[u].pInputRegs        = (tIREG *)  inst->puiIReg;
        mbs->pData->stUnit[u].uiNbrInputRegs    = inst->uiNbrInputRegs;
        mbs->pData->stUnit[0].bInputRegsExtern  = TRUE;
      }

      if (    (inst->puiHReg == NULL)
           && (inst->uiNbrHoldingRegs > 0))
      {
        astatus = TMP_alloc(inst->uiNbrHoldingRegs * sizeof(tHREG),
                            (void **) &pHoldingRegs);
        if (astatus > 0) { inst->uiStatus = astatus; goto END; }
        memset((tHREG *) pHoldingRegs, 0,
               inst->uiNbrHoldingRegs * sizeof(tHREG));
        mbs->pData->stUnit[u].pHoldingRegs = (tHREG *) pHoldingRegs;
        mbs->pData->stUnit[u].uiNbrHoldingRegs = inst->uiNbrHoldingRegs;
      }
      else
      {
        mbs->pData->stUnit[u].pHoldingRegs        = (tHREG *) inst->puiHReg;
        mbs->pData->stUnit[u].uiNbrHoldingRegs    = inst->uiNbrHoldingRegs;
        mbs->pData->stUnit[0].bHoldingRegsExtern  = TRUE;
      }

      inst->uiNbrAllocUnits = inst->uiNbrAllocUnits + 1;

      /* if external mapping is used, only one mapping is allowed */
      if (extMapping == TRUE)
      {
        break;
      }
    }

    mbs->uiPort       = inst->uiPort;
    mbs->uiStep       = INIT;
    mbs->uiReturnStep = INIT;
    mbs->usiCltNr = 0;

    for (i = 0; i < MAX_CLIENT; i++)
    {
      mbs->TOFRecv[i].IN = TRUE;                       /* reset timer */
      TOF(&(mbs->TOFRecv[i]));
    }

    inst->udiIdent = (UDINT) mbs;
    if (inst->uiStatus == ERR_FUB_BUSY)                 /* alloc OK */
    {
      inst->uiNbrAllocUnits = inst->uiNbrAllocUnits;
      inst->uiStatus = ERR_OK;
    }
  }
END: ; /* do nothing */
  /*=========================================================================*/
} /* fMBTSOpen */

/*****************************************************************************
 * END OF CODE
 *****************************************************************************/
/*
  Local Variables:
  c-file-style: bsd
  c-basic-offset: 2
  comment-column: 45
  End:
*/
```

#### fMBTSlave.c
```c
/*****************************************************************************
 * Copyright:    B&R Industrie-Automation AG
 *
 * Project:      Library MBTCP
 *
 * Target:       B&R-PCC
 *
 * AR-Version:   B 2.01
 *
 * AS-Version:   V 3.0.71.16.SP01
 *
 * Filename:     fMBTSlave.c
 *
 * Function:     module-description
 *
 * Dependencies: description of all dependencies
 *
 *****************************************************************************
 * History:
 *
 * Version | Date        | Author      | Description
 * --------------------------------------------------------------------------
 *    1.00 | 2008-sep-19 | H.Anderes   | creation
 *****************************************************************************/

/*****************************************************************************
 * includes
 *****************************************************************************/
/* ansi-c import */
/* system import */
/* user defined import */
#include "MBTCP.h"
#include "MBTSlave.h"

/*****************************************************************************
 * type definitions
 *****************************************************************************/

/*****************************************************************************
 * functions
 *****************************************************************************/
/*===========================================================================*/
void fMBTSlave(struct fMBTSlave* inst)
/*----------------------------------------------------------------------------
  Function:

  Modbus/TCP slave (server) function. fMBTSlave() should be called in
  the CYCLIC section of a task after being configured by
  fMBTSOpen(). The server is closed by fMBTSClose(). This server can
  be read from or written to by fMBTMaster() or widely available
  Modbus over TCP programs.

  History:

  Version | Date        | Author      | Description
  --------------------------------------------------------------------------
  1.00    | 2008-sep-19 | H.Anderes   | creation
  2.00    | 2010-okt-04 | H.Anderes   | refactory
  ===========================================================================*/
{
  /* _LOCAL */
  /* _DYNAMIC */
  tstMBT_SVars* mbs;
  UINT i;
  /*=========================================================================*/
  /* check if nil pointer */
  if (inst == NULL)
  {
    inst->uiStatus = mbtERR_NULL_POINTER;
    goto END;
  }
  mbs = (tstMBT_SVars *) inst->udiIdent;

  if (inst->bEnable < TRUE)
  {
    inst->uiStatus = ERR_FUB_ENABLE_FALSE;
  }
  else
  {
    mbs->bEnable = inst->bEnable;
    for(i = 0; i < MAX_CLIENT; i++)          /* timeout setting */
    {
      if (inst->tiRecvDelay > 0)
      {
        mbs->TOFRecv[i].PT = inst->tiRecvDelay;
      }
      else
      {
        mbs->TOFRecv[i].PT = TIMEOUT_MS;
      }
    }
    /* call  fMBTSStates() */
    fMBTSStates(mbs);

    /* copy internal to the fub interface */
    inst->uiStatus          = mbs->uiStatus;
    inst->uiStep            = mbs->uiStep;
    inst->usiClientNbr      = mbs->usiCltNr;
    inst->usiClientServed   = mbs->usiCltServed;
    inst->tiRecvElapsed     = mbs->TOFRecv[mbs->usiCltServed].ET; /* timeout */
    strcpy(inst->usiClientIP, mbs->cltInfo[mbs->usiCltServed].szIp_addr);
    inst->usiUnit           = mbs->stRecvBuf[mbs->usiCltServed].byte[6];
    inst->usiMBFuncCode     = mbs->stRecvBuf[mbs->usiCltServed].byte[7];
   	strcpy(inst->szMsg, mbs->szMsg);
   	inst->stTcpServerStatus = mbs->stTcpServer.status;
   	inst->usiOpenRetries    = mbs->usiOpenRetries;
   	inst->udiRecvCnt        = mbs->udiRecvCnt;
   	inst->udiSendCnt        = mbs->udiSendCnt;
    /* get client information for debugging */
    for(i = 0; i < MAX_CLIENT; i++)
    {
    	 inst->CltInfo[i].udiIdent = mbs->cltInfo[i].udiIdent;
    	 inst->CltInfo[i].usiPort = mbs->cltInfo[i].usiPort;
      strcpy(inst->CltInfo[i].szIp_addr,mbs->cltInfo[i].szIp_addr);
      strcpy(inst->CltInfo[i].szMsg,mbs->cltInfo[i].szMsg);
    }
  }

END: ; /* do nothing */
  /*=========================================================================*/
} /* fMBTSlave */

/*****************************************************************************
 * END OF CODE
 *****************************************************************************/
/*
  Local Variables:
  c-file-style: bsd
  c-basic-offset: 2
  comment-column: 45
  End:
*/
```

#### fMBTSClose.c
```c
/*****************************************************************************
 * Copyright:    B&R Industrie-Automation AG
 *
 * Project:      Library MBTCP
 *
 * Target:       B&R-PCC
 *
 * AR-Version:   B 2.01
 *
 * AS-Version:   V 3.0.71.16.SP01
 *
 * Filename:     fMBTSClose.c
 *
 * Function:     module-description
 *
 * Dependencies: description of all dependencies
 *
 *****************************************************************************
 * History:
 *
 * Version | Date        | Author      | Description
 * ---------------------------------------------------------------------------
 *    1.00 | 2008-sep-19 | H.Anderes   | creation
 *****************************************************************************/

/*****************************************************************************
 * includes
 *****************************************************************************/
/* ansi-c import */
/* system import */
/* user defined import */
#include "MBTCP.h"
#include "MBTSlave.h"

/*****************************************************************************
 * type definitions
 *****************************************************************************/

/*****************************************************************************
 * functions
 *****************************************************************************/
/*===========================================================================*/
void fMBTSClose(struct fMBTSClose* inst)
/*----------------------------------------------------------------------------
  Function:

  Terminates a Modbus/TCP slave (server) and releases allocated
  memory.  fMBTSClose() should be called in the EXIT section of a
  task. See also fMBTSOpen() and fMBTSlave().

  History:

  Version | Date        | Author      | Description
  ----------------------------------------------------------------------------
     1.00 | 2008-sep-19 | H.Anderes    | creation
  ===========================================================================*/
{
  /* _LOCAL */
  UINT u, c, fstatus = 0;
  USINT usiClientNr;
  /* _DYNAMIC */
  tstMBT_SVars* mbs;
  /*=========================================================================*/
  /* check if nil pointer */
  if (inst == NULL)
  {
    inst->uiStatus = mbtERR_NULL_POINTER;
	   goto END;
  }
  mbs = (tstMBT_SVars *)inst->udiIdent;

  if (inst->bEnable < TRUE)
  {
    inst->uiStatus = ERR_FUB_ENABLE_FALSE;
  }
  else
  {
    inst->uiStatus = ERR_FUB_BUSY;

    /* disconnect all clients and close slave's port */
    mbs->uiStep = CLOSE_SLAVE;
    usiClientNr = mbs->usiCltNr;
    /* call fMBTSStates() */
    fMBTSStates(mbs);  /* internal main state machine */
    c = 0;
    while (    (mbs->bClosing > 0)
            && (c < MAX_CLOSE_LOOPS))
    {
      fMBTSStates(mbs);
      c++;
    }

    for (u = 0; u < mbs->pData->uiNbrUnits; u++)
    {
      if (mbs->pData->stUnit[0].bCoilsExtern == FALSE)
      {
        fstatus = TMP_free(mbs->pData->stUnit[u].uiNbrCoils * sizeof(tCOIL),
                             (void**)(mbs->pData->stUnit[u].pCoils));
        if (fstatus > 0)
        {
          inst->uiStatus = fstatus;
          ERRxwarning(fstatus, 0,
                      (STRING*)"fMBTSClose: failed to TMP_free pCoils");
          goto END;  /* EXIT_FAILURE; */
        }
      }

      if (mbs->pData->stUnit[0].bDiscreteInputsExtern == FALSE)
      {
        fstatus =
          TMP_free(mbs->pData->stUnit[u].uiNbrDiscreteInputs * sizeof(tDINP),
                   (void**)(mbs->pData->stUnit[u].pDiscreteInputs));
        if (fstatus > 0)
        {
          inst->uiStatus = fstatus;
          ERRxwarning(fstatus, 0,
                      (STRING*)"fMBTSClose: failed to TMP_free pDiscreteInputs");
          goto END;  /* EXIT_FAILURE; */
        }
      }

      if (mbs->pData->stUnit[0].bInputRegsExtern == FALSE)
      {
        fstatus = TMP_free(mbs->pData->stUnit[u].uiNbrInputRegs * sizeof(tIREG),
                           (void**)(mbs->pData->stUnit[u].pInputRegs));
        if (fstatus > 0)
        {
          inst->uiStatus = fstatus;
          ERRxwarning(fstatus, 0,
                      (STRING*)"fMBTSClose: failed to TMP_free pInputRegs");
          goto END;  /* EXIT_FAILURE; */
        }
      }

      if (mbs->pData->stUnit[0].bHoldingRegsExtern == FALSE)
      {
        fstatus = TMP_free(mbs->pData->stUnit[u].uiNbrHoldingRegs * sizeof(tHREG),
                           (void**)(mbs->pData->stUnit[u].pHoldingRegs));
        if (fstatus > 0)
        {
          inst->uiStatus = fstatus;
          ERRxwarning(fstatus, 0,
                      (STRING*)"fMBTSClose: failed to TMP_free pHoldingRegs");
          goto END;  /* EXIT_FAILURE; */
        }
      }
    }

    fstatus = TMP_free(sizeof(tstMBT_SData), (void**)mbs->pData);
    if (fstatus > 0)
    {
      inst->uiStatus = fstatus;
      ERRxwarning(fstatus, 0,
                  (STRING*)"fMBTSClose: failed to TMP_free pData");
        goto END;  /* EXIT_FAILURE; */
    }
    fstatus = TMP_free(sizeof(tstMBT_SVars), (void**)mbs);
    if (fstatus > 0)
    {
      inst->uiStatus = fstatus;
      ERRxwarning(fstatus, 0, (STRING*)"fMBTSClose: failed to TMP_free mbs");
      goto END;  /* EXIT_FAILURE; */
    }
  }
  END: ; /* do nothing */
  /*=========================================================================*/
  } /* fMBTSClose */

/*****************************************************************************
 * END OF CODE
 *****************************************************************************/
/*
Local Variables:
c-file-style: bsd
c-basic-offset: 2
comment-column: 45
End:
 */
```

#### fMBTSRW.c
```c
/*****************************************************************************
 * Copyright:    B&R Industrie-Automation AG
 *
 * Project:      Library MBTCP
 *
 * Target:       B&R-PCC
 *
 * AR-Version:   B 2.01
 *
 * AS-Version:   V 3.0.71.16.SP01
 *
 * Filename:     fMBTSRW.c
 *
 * Function:     module-description
 *
 * Dependencies: description of all dependencies
 *
 *****************************************************************************
 * History:
 *
 * Version | Date        | Author      | Description
 * --------------------------------------------------------------------------
 *    1.00 | 2008-sep-25 | H.Anderes    | creation
 *****************************************************************************/

/*****************************************************************************
 * includes
 *****************************************************************************/
/* ansi-c import */
/* system import */
/* user defined import */
#include "MBTCP.h"
#include "MBTSlave.h"

/*****************************************************************************
 * type definitions
 *****************************************************************************/

/*****************************************************************************
 * functions
 *****************************************************************************/
/*===========================================================================*/
void fMBTSRW(struct fMBTSRW* inst)
/*---------------------------------------------------------------------------
  Function:
  <header>
  <p>
   Read/write individual values from/to coils and registers of given unit.
   The function code to use in member uiFcode of the passed structure is the
   same as for Modbus (0x01..0x06) and two user defined functions (0x41,0x42).
   See Modbus function codes.

  History:

  Version | Date        | Author      | Description
  --------------------------------------------------------------------------
  1.00 | 2008-sep-19 | H.Anderes    | creation
  1.01 | 2009-mar-03 | H.Anderes   | implementation FC15, FC16
  1.01 | 2009-dez-09 | H.Anderes   | implementation FC23, change FUB interface
  ===========================================================================*/
{
  /* _LOCAL */
  UINT u, i;
  UINT coil;
  UINT hreg;
  UINT ireg;
  /* _DYNAMIC */
  tstMBT_SVars* mbs;
  tCOIL* pCoilVal;
  tDINP* pDInpVal;
  tIREG* pIRegVal;
  tHREG* pHRegVal;
  /*=========================================================================*/
  /* check if nil pointer */
  if (inst == NULL)
  {
    inst->uiStatus = mbtERR_NULL_POINTER;
	   goto END;
  }
  mbs = (tstMBT_SVars *) inst->udiIdent;

  if (inst->bEnable < TRUE)
  {
    inst->uiStatus = ERR_FUB_ENABLE_FALSE;
  }
  else
  {
    inst->uiStatus = ERR_FUB_BUSY;

    u = inst->usiUnit;
    if (    (u >= mbs->pData->uiNbrUnits + mbs->pData->uiOffsetUnits)
         || (u < mbs->pData->uiOffsetUnits))
      { inst->uiStatus = mbtERR_NBR_UNITS; goto END; }

    switch(inst->usiFCode)
    {
    /*------------------------------------------------------------------------
      READ: read coils
    -------------------------------------------------------------------------*/
    case MBT_READ_COILS:                     /* 0x01 */
      if (inst->puiReadVal == NULL)
        { inst->uiStatus = mbtERR_DATA_ADDRESS; goto END; }
      pCoilVal = (tCOIL*) inst->puiReadVal;
      i = inst->uiReadAddr;
      if (i > mbs->pData->stUnit[u].uiNbrCoils)
        { inst->uiStatus = mbtERR_DATA_ADDRESS; goto END; }
      if (    (inst->uiReadQty > 0)
           && (inst->uiReadQty <= (*(mbs->pData)).stUnit[u].uiNbrCoils))
      {
        if (    (inst->uiReadAddr + inst->uiReadQty)
             <= (*(mbs->pData)).stUnit[u].uiNbrCoils)
        {
          for (i = 0; i < inst->uiReadQty; i++)
          {
            coil = inst->uiReadAddr + i;
            if(((*(mbs->pData)).stUnit[u].pCoils[(i)] & (USINT)(0x01)))
              pCoilVal[(i)*2 + BYTE_OFFSET]  = (tCOIL) 1;
            else
              pCoilVal[(i)*2 + BYTE_OFFSET]  = (tCOIL) 0;
           }
        }
      }
      break;
	   /*-------------------------------------------------------------------------
      READ: read discrete inputs
    --------------------------------------------------------------------------*/
    case MBT_READ_DISCRETE_INPUTS:           /* 0x02 */
     if (inst->puiReadVal == NULL)
        { inst->uiStatus = mbtERR_DATA_ADDRESS; goto END; }
      pDInpVal = (tDINP*) inst->puiReadVal;
      i = inst->uiReadAddr;
      if (i > mbs->pData->stUnit[u].uiNbrDiscreteInputs)
        { inst->uiStatus = mbtERR_DATA_ADDRESS; goto END; }
      if (   (inst->uiReadQty > 0)
          && (inst->uiReadQty <= (*(mbs->pData)).stUnit[u].uiNbrDiscreteInputs))
      {
        if (    (inst->uiReadAddr + inst->uiReadQty)
             <= (*(mbs->pData)).stUnit[u].uiNbrDiscreteInputs)
        {
          for (i = 0; i < inst->uiReadQty; i++)
          {
            coil = inst->uiReadAddr + i;
            if(((*(mbs->pData)).stUnit[u].pDiscreteInputs[(i)] & (USINT)(0x01)))
              pDInpVal[(i)*2 + BYTE_OFFSET]  = (tCOIL) 1;
            else
              pDInpVal[(i)*2 + BYTE_OFFSET]  = (tCOIL) 0;
           }
        }
      }
      break;
	   /*--------------------------------------------------------------------------
      READ: read discrete inputs
    ---------------------------------------------------------------------------*/
    case MBT_READ_HOLDING_REGISTERS:         /* 0x03 */
      if (inst->puiReadVal == NULL)
        { inst->uiStatus = mbtERR_DATA_ADDRESS; goto END; }
      pHRegVal = (tHREG*) inst->puiReadVal;
      i = inst->uiReadAddr;
      if (i > mbs->pData->stUnit[u].uiNbrHoldingRegs)
        { inst->uiStatus = mbtERR_DATA_ADDRESS; goto END; }
      if (    (inst->uiReadQty > 0)
           && (inst->uiReadQty <= (*(mbs->pData)).stUnit[u].uiNbrHoldingRegs))
      {
        if (    (inst->uiReadAddr + inst->uiReadQty)
             <= (*(mbs->pData)).stUnit[u].uiNbrHoldingRegs)
        {
          for (i = 0; i < inst->uiReadQty; i++)
          {
            hreg = inst->uiReadAddr + i;
            pHRegVal[(i)] = mbs->pData->stUnit[u].pHoldingRegs[hreg];
          }
        }
      }
      break;
	   /*--------------------------------------------------------------------------
      READ: read input registers
    ---------------------------------------------------------------------------*/
    case MBT_READ_INPUT_REGISTERS:           /* 0x04 */
      if (inst->puiReadVal == NULL)
        { inst->uiStatus = mbtERR_DATA_ADDRESS; goto END; }
      pIRegVal = (tIREG*) inst->puiReadVal;
      i = inst->uiReadAddr;
      if (i > mbs->pData->stUnit[u].uiNbrInputRegs)
        { inst->uiStatus = mbtERR_DATA_ADDRESS; goto END; }
      if (    (inst->uiReadQty > 0)
           && (inst->uiReadQty <= (*(mbs->pData)).stUnit[u].uiNbrInputRegs))
        {
          if (    (inst->uiReadAddr + inst->uiReadQty)
               <= (*(mbs->pData)).stUnit[u].uiNbrInputRegs)
          {
            for (i = 0; i < inst->uiReadQty; i++)
            {
              ireg = inst->uiReadAddr + i;
              pIRegVal[(i)] = mbs->pData->stUnit[u].pInputRegs[ireg];
            }
          }
        }
      break;
	   /*--------------------------------------------------------------------------
      WRITE: write single coil
    ---------------------------------------------------------------------------*/
    case MBT_WRITE_SINGLE_COIL:              /* 0x05 */
     if (inst->puiWriteVal == NULL)
        { inst->uiStatus = mbtERR_DATA_ADDRESS; goto END; }
      pCoilVal = (tCOIL*) inst->puiWriteVal+BYTE_OFFSET;
      i = inst->uiWriteAddr;
      if (i > mbs->pData->stUnit[u].uiNbrCoils)
        { inst->uiStatus = mbtERR_DATA_ADDRESS; goto END; }
      mbs->pData->stUnit[u].pCoils[i] = *pCoilVal;
      break;
	   /*--------------------------------------------------------------------------
      WRITE: write single register
    ---------------------------------------------------------------------------*/
    case MBT_WRITE_SINGLE_REGISTER:          /* 0x06 */
      if (inst->puiWriteVal == NULL)
        { inst->uiStatus = mbtERR_DATA_ADDRESS; goto END; }
      pHRegVal = (tHREG*) inst->puiWriteVal;
      i = inst->uiWriteAddr;
   	  if (i > mbs->pData->stUnit[u].uiNbrHoldingRegs)
           { inst->uiStatus = mbtERR_DATA_ADDRESS; goto END; }
       mbs->pData->stUnit[u].pHoldingRegs[i] = *pHRegVal;
 	    break;
	   /*--------------------------------------------------------------------------
      WRITE: write discrete inputs
    ---------------------------------------------------------------------------*/
 	  case BR_MBT_WRITE_DISCRETE_INPUTS:       /* 0x41 */
      if (inst->puiWriteVal == NULL)
        { inst->uiStatus = mbtERR_DATA_ADDRESS; goto END; }
      pDInpVal = (tDINP*) inst->puiWriteVal;
      i = inst->uiWriteAddr;
   	  if (i > mbs->pData->stUnit[u].uiNbrDiscreteInputs)
           { inst->uiStatus = mbtERR_DATA_ADDRESS; goto END; }
      if (    (inst->uiWriteQty > 0)
            && (inst->uiWriteQty <= (*(mbs->pData)).stUnit[u].uiNbrDiscreteInputs))
      {
        if (    (inst->uiWriteAddr + inst->uiWriteQty)
             <= (*(mbs->pData)).stUnit[u].uiNbrDiscreteInputs)
        {
           for (i = 0; i < inst->uiWriteQty; i++)
           {
             coil = inst->uiWriteAddr + i;

             if((pDInpVal[(i*2)+ BYTE_OFFSET] & (USINT)(0x01)))
                 (*(mbs->pData)).stUnit[u].pDiscreteInputs[coil] = (tCOIL) 1;
             else
                 (*(mbs->pData)).stUnit[u].pDiscreteInputs[coil] = (tCOIL) 0;
            }
        }
      }
 	    break;
	  	/*--------------------------------------------------------------------------
      WRITE: write input register
    ---------------------------------------------------------------------------*/
 	  case BR_MBT_WRITE_INPUT_REGISTERS:        /* 0x42 */
      if (inst->puiWriteVal == NULL)
        { inst->uiStatus = mbtERR_DATA_ADDRESS; goto END; }
      pIRegVal = (tIREG*) inst->puiWriteVal;
      i = inst->uiWriteAddr;
   	  if (i > mbs->pData->stUnit[u].uiNbrInputRegs)
           { inst->uiStatus = mbtERR_DATA_ADDRESS; goto END; }
      if (   (inst->uiWriteQty > 0)
          && (inst->uiWriteQty <= (*(mbs->pData)).stUnit[u].uiNbrInputRegs))
       {
        if (   (inst->uiWriteAddr + inst->uiWriteQty)
            <= (*(mbs->pData)).stUnit[u].uiNbrInputRegs)
        {
          for (i = 0; i < inst->uiWriteQty; i++)
          {
            ireg = inst->uiWriteAddr + i;
            (*(mbs->pData)).stUnit[u].pInputRegs[ireg] = pIRegVal[(i)];
          }
        }
      }
      break;
	  	/*-------------------------------------------------------------------------
      WRITE: write multiple coils
    --------------------------------------------------------------------------*/
    case MBT_WRITE_MULTIPLE_COILS:           /* 0x0F */
      if (inst->puiWriteVal == NULL)
        { inst->uiStatus = mbtERR_DATA_ADDRESS; goto END; }
      pCoilVal = (tCOIL*) inst->puiWriteVal;
      i = inst->uiWriteAddr;
      if (i > mbs->pData->stUnit[u].uiNbrCoils)
        { inst->uiStatus = mbtERR_DATA_ADDRESS; goto END; }
    		if (    (inst->uiWriteQty > 0)
    	      && (inst->uiWriteQty <= (*(mbs->pData)).stUnit[u].uiNbrCoils))
    		{
  	    	if (    (inst->uiWriteAddr + inst->uiWriteQty)
  	         	<= (*(mbs->pData)).stUnit[u].uiNbrCoils)
  	    	{
  	        for (i = 0; i < inst->uiWriteQty; i++)
  	      		{
  	          coil = inst->uiWriteAddr + i;

  						     if((pCoilVal[(i)*2+BYTE_OFFSET]& (USINT)(0x01)))
  		          			(*(mbs->pData)).stUnit[u].pCoils[coil] = (tCOIL) 1;
  		        	else
  		          			(*(mbs->pData)).stUnit[u].pCoils[coil] = (tCOIL) 0;
  			       }
  		     }
    		}
		   break;
    /*--------------------------------------------------------------------------
      WRITE: write multiple register
    ---------------------------------------------------------------------------*/
    case MBT_WRITE_MULTIPLE_REGISTERS:       /* 0x10 */
      if (inst->puiWriteVal == NULL)
        { inst->uiStatus = mbtERR_DATA_ADDRESS; goto END; }
      pHRegVal = (tHREG*) inst->puiWriteVal;
      i = inst->uiWriteAddr;
      if (i > mbs->pData->stUnit[u].uiNbrHoldingRegs)
        { inst->uiStatus = mbtERR_DATA_ADDRESS; goto END; }
    		if (    (inst->uiWriteQty > 0)
          	&& (inst->uiWriteQty <= (*(mbs->pData)).stUnit[u].uiNbrHoldingRegs))
      		{
    		   if (   (inst->uiWriteAddr + inst->uiWriteQty)
    		       <= (*(mbs->pData)).stUnit[u].uiNbrHoldingRegs)
    		   {
    		     for (i = 0; i < inst->uiWriteQty; i++)
    		     {
    				     hreg = inst->uiWriteAddr + i;
    		       (*(mbs->pData)).stUnit[u].pHoldingRegs[hreg] = pHRegVal[(i)];
    		     }
    		   }
    		}
	     break;
    /*--------------------------------------------------------------------------
      WRITE: read and write multiple register
    ---------------------------------------------------------------------------*/
    case READ_WRITE_MULTIPLE_REGISTERS:
      /*****************write multiple register ***************/
      if (inst->puiWriteVal == NULL)
        { inst->uiStatus = mbtERR_DATA_ADDRESS; goto END; }
      pHRegVal = (tHREG*) inst->puiWriteVal;
      i = inst->uiWriteAddr;
      if (i > mbs->pData->stUnit[u].uiNbrHoldingRegs)
        { inst->uiStatus = mbtERR_DATA_ADDRESS; goto END; }
      if (    (inst->uiWriteQty > 0)
           && (inst->uiWriteQty <= (*(mbs->pData)).stUnit[u].uiNbrHoldingRegs))
        {
          if (   (inst->uiWriteAddr + inst->uiWriteQty)
              <= (*(mbs->pData)).stUnit[u].uiNbrHoldingRegs)
          {
            for (i = 0; i < inst->uiWriteQty; i++)
            {
              hreg = inst->uiWriteAddr + i;
              (*(mbs->pData)).stUnit[u].pHoldingRegs[hreg] = pHRegVal[(i)];
            }
          }
        }
      /*****************read multiple register ***************/
     if ( inst->puiReadVal == NULL)
        { inst->uiStatus = mbtERR_DATA_ADDRESS; goto END; }
      pHRegVal = (tHREG*) inst->puiReadVal;
      i = inst->uiReadAddr;
      if (i > mbs->pData->stUnit[u].uiNbrHoldingRegs)
        { inst->uiStatus = mbtERR_DATA_ADDRESS; goto END; }
      if (    (inst->uiReadQty > 0)
           && (inst->uiReadQty <= (*(mbs->pData)).stUnit[u].uiNbrHoldingRegs))
        {
          if (    (inst->uiReadAddr + inst->uiReadQty)
               <= (*(mbs->pData)).stUnit[u].uiNbrHoldingRegs)
          {
            for (i = 0; i < inst->uiReadQty; i++)
            {
              hreg = inst->uiReadAddr + i;
              pHRegVal[(i)] = mbs->pData->stUnit[u].pHoldingRegs[hreg];
            }
          }
        }
      break;
    default:
      { inst->uiStatus = mbtERR_ILLEGAL_FUNCTION; goto END; }
    }
    inst->uiStatus = ERR_OK;
  }
END: ; /* do nothing */
  /*=========================================================================*/
} /* fMBTSRW */

/*****************************************************************************
 * END OF CODE
 *****************************************************************************/
/*
  Local Variables:
  c-file-style: bsd
  c-basic-offset: 2
  comment-column: 45
  End:
*/
```

#### fMBTSFill.c
```c
/*****************************************************************************
 * Copyright:    B&R Industrie-Automation AG
 *
 * Project:      Library MBTCP
 *
 * Target:       B&R-PCC
 *
 * AR-Version:   B 2.01
 *
 * AS-Version:   V 3.0.71.16.SP01
 *
 * Filename:     fMBTSFill.c
 *
 * Function:     module-description
 *
 * Dependencies: description of all dependencies
 *
 *****************************************************************************
 * History:
 *
 * Version | Date        | Author      | Description
 * --------------------------------------------------------------------------
 *    1.00 | 2008-sep-19 | H.Anderes    | creation
 *****************************************************************************/

/*****************************************************************************
 * includes
 *****************************************************************************/
/* ansi-c import */
/* system import */
/* user defined import */
#include "MBTCP.h"
#include "MBTSlave.h"

/*****************************************************************************
 * type definitions
 *****************************************************************************/

/*****************************************************************************
 * functions
 *****************************************************************************/
/*===========================================================================*/
void fMBTSFill(struct fMBTSFill* inst)
/*---------------------------------------------------------------------------
  Function:

  Initialize the slave's data units (coils and registers) with
  values. Coils and Discrete Inputs are initialized with 0, 1,
  0... Input registers are filled with 1000, 1001, 1002... Holding
  registers are initialized with 0, 1, 2...

  History:

  Version | Date        | Author      | Description
  --------------------------------------------------------------------------
     1.00 | 2008-sep-19 | H.Anderes    | creation
  ===========================================================================*/
  {
  /* _LOCAL */
  UINT u, i, imax;
  /* _DYNAMIC */
  tstMBT_SVars* mbs;
  /*=========================================================================*/
  /* check if nil pointer */
  if (inst == NULL)
    {
    inst->uiStatus = mbtERR_NULL_POINTER;
	goto END;
    }
  mbs = (tstMBT_SVars *) inst->udiIdent;

  if (inst->bEnable < TRUE)
  {
    inst->uiStatus = ERR_FUB_ENABLE_FALSE;
  }
  else
  {
    inst->uiStatus = ERR_FUB_BUSY;

    for (u = mbs->pData->uiOffsetUnits; u < (mbs->pData->uiNbrUnits + mbs->pData->uiOffsetUnits); u++)
    {
      imax = mbs->pData->stUnit[u].uiNbrCoils;
      for (i = 0; i < imax; i++) {
        mbs->pData->stUnit[u].pCoils[i] = 0;
        mbs->pData->stUnit[u].pCoils[i] = (tCOIL)(i & 0x0001);
      }
      imax = mbs->pData->stUnit[u].uiNbrDiscreteInputs;
      for (i = 0; i < imax; i++) {
        mbs->pData->stUnit[u].pDiscreteInputs[i] = 0;
        mbs->pData->stUnit[u].pDiscreteInputs[i] = (tDINP)(i & 0x0001);
      }
      imax = mbs->pData->stUnit[u].uiNbrInputRegs;
      for (i = 0; i < imax; i++) {
        mbs->pData->stUnit[u].pInputRegs[i] = (tIREG)(1000 + i);
      }
      imax = mbs->pData->stUnit[u].uiNbrHoldingRegs;
      for (i = 0; i < imax; i++) {
        mbs->pData->stUnit[u].pHoldingRegs[i] = (tHREG)(i);
      }
    }
    mbs->bEnable = TRUE;
    inst->uiStatus = ERR_OK;
  }
  END: ; /* do nothing */
  /*=========================================================================*/
  } /* fMBTSFill */

/*****************************************************************************
 * END OF CODE
 *****************************************************************************/
```

#### fMBTMOpen.c
```c
/*****************************************************************************
 * Copyright:    B&R Industrie-Automation AG
 *
 * Project:      Library MBTCP
 *
 * Target:       B&R-PCC
 *
 * AR-Version:   B 2.01
 *
 * AS-Version:   V 3.0.71.16.SP01
 *
 * Filename:     fMBTMOpen.c
 *
 * Function:     module-description
 *
 * Dependencies: description of all dependencies
 *
 *****************************************************************************
 * History:
 *
 * Version | Date        | Author      | Description
 * ---------------------------------------------------------------------------
 *    1.00 | 2008-Oct-01 | H.Anderes    | creation
 *****************************************************************************/

/*****************************************************************************
 * includes
 *****************************************************************************/
/* ansi-c import */
/* system import */
/* user defined import */
#include "MBTCP.h"
#include "MBTMaster.h"

/*****************************************************************************
 * type definitions
 *****************************************************************************/

/*****************************************************************************
 * functions
 *****************************************************************************/
/*==========================================================================*/
void fMBTMOpen(struct fMBTMOpen* inst)
/*---------------------------------------------------------------------------
  Function:

  Allocates memory and pre-configures Modbus TCP Master.
  fMBTMOpen() should be called in the INIT section of a task prior
  to fMBTMaster(). See also fMBTMClose() to close the master in the
  task's EXIT section. The master connects to the Modbus TCP slave
  available at the IP address provided by szSlvIPAddr.

  History:

  Version | Date        | Author      | Description
  ---------------------------------------------------------------------------
     1.00 | 2008-Oct-01 | H.Anderes    | creation
  ===========================================================================*/
  {
  /* _LOCAL */
  UINT astatus = 0;
  RTInfo_typ stRTInfo;
  UDINT udiCycleTime;

  /* _DYNAMIC */
  tstMBT_MVars *mbm;
  tstMBT_MData *pData;

  /*=========================================================================*/
  if (inst == NULL)
  {
    inst->uiStatus = mbtERR_NULL_POINTER;
    goto END;
  }
  if (inst->bEnable < TRUE)
  {
    inst->uiStatus = ERR_FUB_ENABLE_FALSE;
  }
  else
  {
    inst->uiStatus = ERR_FUB_BUSY;
    if (inst->szSlvIPAddr == NULL)
    {
      inst->uiStatus = mbtERR_IP_ADRESS;
      goto END;
    }

    astatus = TMP_alloc(sizeof(tstMBT_MVars), (void**)&mbm);
    if (astatus > 0) { inst->uiStatus = astatus; goto END; }
    memset(mbm, 0, sizeof(tstMBT_MVars));
    astatus = TMP_alloc(sizeof(tstMBT_MData), (void**)&pData);
    if (astatus > 0) { inst->uiStatus = astatus; goto END; }
    memset(pData, 0, sizeof(tstMBT_MData));
    mbm->pData = pData;

    stRTInfo.enable = TRUE;
    RTInfo(&stRTInfo);
    udiCycleTime = (UDINT)(stRTInfo.cycle_time / 1000);
    stRTInfo.enable = FALSE;
    /* call RTInfo() */
    RTInfo(&stRTInfo);

    if (inst->uiPort < 1)
    {
      inst->uiPort = MBT_SLAVE_PORT;
    }
    if (inst->uiRecvTimeout < 1)
    {
      inst->uiRecvTimeout = RECV_TIMEOUT_DFLT;
    }

    memmove(&(mbm->slvIPAddr),&(inst->szSlvIPAddr), IPADDR_L);
    mbm->uiPort 	      = inst->uiPort;
    mbm->udiCycleTime	 = udiCycleTime;
    mbm->uiRecvTimeout = inst->uiRecvTimeout;
    mbm->uiStep		      = INIT;

    inst->udiIdent = (UDINT) mbm;
    if (inst->uiStatus == ERR_FUB_BUSY)         /* alloc OK */
    {
      inst->uiStatus = ERR_OK;
    }
  }
  END: ; /* do nothing */
  /*=========================================================================*/
  } /* fMBTMOpen */

/*****************************************************************************
 * END OF CODE
 *****************************************************************************/
 /*
Local Variables:
c-file-style: bsd
c-basic-offset: 2
comment-column: 45
End:
 */
```

#### fMBTMaster.c
```c
/****************************************************************************
 * Copyright:    B&R Industrie-Automation AG
 *
 * Project:      Library MBTCP
 *
 * Target:       B&R-PCC
 *
 * AR-Version:   B 2.01
 *
 * AS-Version:   V 3.0.71.16.SP01
 *
 * Filename:     fMBTMaster.c
 *
 * Function:     module-description
 *
 * Dependencies: description of all dependencies
 *
 ****************************************************************************
 * History:
 *
 * Version | Date        | Author      | Description
 * --------------------------------------------------------------------------
 *    1.00 | 2008-Oct-03 | H.Anderes    | creation
 *****************************************************************************/

/*****************************************************************************
 * includes
 *****************************************************************************/
/* ansi-c import */
/* system import */
/* user defined import */
#include "MBTCP.h"
#include "MBTMaster.h"

/*****************************************************************************
 * type definitions
 *****************************************************************************/

/*****************************************************************************
 * functions
 *****************************************************************************/
/*===========================================================================*/
void fMBTMaster(struct fMBTMaster* inst)
/*---------------------------------------------------------------------------
  Function:

  Modbus/TCP master (client) function. fMBTMaster()
  should be called in the CYCLIC section of a task after being
  configured by fMBTMOpen(). The master is closed by fMBTMClose().
  This master writes to or reads from a slave running fMBTSlave() or
  other widely available Modbus over TCP slave programs.

  History:

  Version | Date        | Author      | Description
  --------------------------------------------------------------------------
  1.00    | 2008-Oct-03 | H.Anderes    | creation
  ===========================================================================*/
{
  /* _LOCAL */
  /* _DYNAMIC */
  tstMBT_MVars *mbm;
  /*=========================================================================*/
  if (inst == NULL)
  {
    inst->uiStatus = mbtERR_NULL_POINTER;
    goto END;
  }
  mbm = (tstMBT_MVars *) inst->udiIdent;

  if (inst->bEnable < TRUE)
  {
    inst->uiStatus = ERR_FUB_ENABLE_FALSE;
  }
  else
  {

    mbm->bEnable = inst->bEnable;
    /* call fMBTMStates */
    fMBTMStates(mbm);

    inst->uiStep        = mbm->uiStep;
    inst->uiTxID        = mbm->uiTxID;
    inst->usiMBFuncCode = mbm->usiRecvBuf[7];
    inst->usiRxByteCnt  = mbm->usiRecvBuf[8];
	   strcpy(inst->szMsg,mbm->szMsg);
    inst->uiStatus      = mbm->uiStatus;
}

END: ; /* do nothing */
  /*=========================================================================*/
} /* fMBTMaster */

/*****************************************************************************
 * END OF CODE
 *****************************************************************************/
/*
  Local Variables:
  c-file-style: bsd
  c-basic-offset: 2
  comment-column: 45
  End:
 */
```

#### fMBTMClose.c
```c
/****************************************************************************
 * Copyright:    B&R Industrie-Automation AG
 *
 * Project:      Library MBTCP
 *
 * Target:       B&R-PCC
 *
 * AR-Version:   B 2.01
 *
 * AS-Version:   V 3.0.71.16.SP01
 *
 * Filename:     fMBTMClose.c
 *
 * Function:     module-description
 *
 * Dependencies: description of all dependencies
 *
 ****************************************************************************
 * History:
 *
 * Version | Date        | Author      | Description
 * --------------------------------------------------------------------------
 *    1.00 | 2008-Oct-03 | H.Anderes    | creation
 *****************************************************************************/

/*****************************************************************************
 * includes
 *****************************************************************************/
/* ansi-c import */
/* system import */
/* user defined import */
#include "MBTCP.h"
#include "MBTMaster.h"

/*****************************************************************************
 * type definitions
 *****************************************************************************/

/*****************************************************************************
 * functions
 *****************************************************************************/
/*===========================================================================*/
void fMBTMClose(struct fMBTMClose* inst)
/*---------------------------------------------------------------------------
  Function:

  Terminates a Modbus/TCP master (client) and releases allocated memory.
  fMBTMClose() should be called in the EXIT section of a task.
  See also fMBTMOpen() and fMBTMaster().

  History:

  Version | Date        | Author      | Description
  --------------------------------------------------------------------------
  1.00 | 2008-Oct-03 | H.Anderes    | creation
  ===========================================================================*/
{
  /* _LOCAL */
  UINT fstatus = 0;
  USINT i;
  /* _DYNAMIC */
  tstMBT_MVars *mbm;
  /*=========================================================================*/
  if (inst == NULL)
  {
    inst->uiStatus = mbtERR_NULL_POINTER;
    goto END;
  }
  mbm = (tstMBT_MVars *) inst->udiIdent;

  if (inst->bEnable < TRUE)
  {
    inst->uiStatus = ERR_FUB_ENABLE_FALSE;
  }
  else
  {
    inst->uiStatus = ERR_FUB_BUSY;

    /* disconnect from slave */
    mbm->uiStep = CLOSE_PORT;
    for (i = 0; i < 2; i++)                  /* 2 iterations needed */
      fMBTMStates(mbm);

    fstatus = TMP_free(sizeof(tstMBT_MData), (void**)mbm->pData);
    if (fstatus > 0)
    {
      inst->uiStatus = fstatus;
      ERRxwarning(fstatus, 0, (STRING*)"fMBTMClose: failed to TMP_free pData");
        goto END;
    }
    fstatus = TMP_free(sizeof(tstMBT_MVars), (void**)mbm);
    if (fstatus > 0)
    {
      inst->uiStatus = fstatus;
      ERRxwarning(fstatus, 0, (STRING*)"fMBTMClose: failed to TMP_free mbm");
      goto END;
    }
  }

END: ; /* do nothing */
  /*=========================================================================*/
} /* fMBTMClose */

/*****************************************************************************
 * END OF CODE
 *****************************************************************************/

/*
  Local Variables:
  c-file-style: bsd
  c-basic-offset: 2
  comment-column: 45
  End:
*/
```

#### fMBTMRW.c
```c
/*****************************************************************************
 * Copyright:    B&R Industrie-Automation AG
 *
 * Project:      Library MBTCP
 *
 * Target:       B&R-PCC
 *
 * AR-Version:   B 2.01
 *
 * AS-Version:   V 3.0.71.16.SP01
 *
 * Filename:     fMBTMRW.c
 *
 * Function:     module-description
 *
 * Dependencies: description of all dependencies
 *
 *****************************************************************************
 * History:
 *
 * Version | Date        | Author      | Description
 * --------------------------------------------------------------------------
 *    1.00 | 2008-Oct-03 | H.Anderes    | creation
 *****************************************************************************/

/*****************************************************************************
 * includes
 *****************************************************************************/
/* ansi-c import */
/* system import */
/* user defined import */
#include "MBTCP.h"
#include "MBTMaster.h"

/*****************************************************************************
 * type definitions
 *****************************************************************************/

/*****************************************************************************
 * functions
 *****************************************************************************/
/*===========================================================================*/
void fMBTMRW(struct fMBTMRW* inst)
/*---------------------------------------------------------------------------
  Function:

  Read/write individual values from/to coils and registers of given unit.
  The function code to use in member uiFcode of the passed structure is the
  same as for Modbus (0x01..0x06).

  History:

  Version | Date        | Author      | Description
  --------------------------------------------------------------------------
  1.00 | 2008-Oct-06 | H.Anderes    | creation
  ===========================================================================*/
{
  /* _LOCAL */
  /* _DYNAMIC */
  tstMBT_MVars* mbm;
  /*=========================================================================*/
  /* check if nil pointer */
  if (inst == NULL)
  {
    inst->uiStatus = mbtERR_NULL_POINTER;
	goto END;
  }
  mbm = (tstMBT_MVars *) inst->udiIdent;

  if (inst->bEnable < TRUE)
  {
    inst->uiStatus = ERR_FUB_ENABLE_FALSE;
  }
  else
  {
    inst->uiStatus = ERR_FUB_BUSY;

    mbm->pData->actParam[0].usiFCode	  = inst->usiFCode;
    mbm->pData->actParam[0].usiUnit 	  = inst->usiUnit;
    mbm->pData->actParam[0].uiReadAddr  = inst->uiReadAddr;
    mbm->pData->actParam[0].uiReadQty 	= inst->uiReadQty;
    mbm->pData->actParam[0].uiWriteAddr = inst->uiWriteAddr;
    mbm->pData->actParam[0].uiWriteQty  = inst->uiWriteQty;

    if (inst->bPoll)
    {
      mbm->pData->actEnable[0].bCyclic 	= TRUE;
      mbm->pData->actEnable[0].bSingle 	= FALSE;
      mbm->pData->actParam[0].udiTimer 	= inst->udiPollPeriod;
    }
    else
    {
      mbm->pData->actEnable[0].bCyclic 	= FALSE;
      mbm->pData->actEnable[0].bSingle 	= TRUE;
      mbm->pData->actParam[0].udiTimer 	= 0;
    }

    switch(inst->usiFCode)
    {
    case MBT_READ_COILS:                     /* 0x01 */
    case MBT_READ_DISCRETE_INPUTS:           /* 0x02 */
       if (inst->uiReadQty > MAX_COILS)
         { inst->uiStatus = mbtERR_MAX_NBR_COILS; inst->bRecvOK = FALSE; goto END; }
      break;
    case MBT_READ_HOLDING_REGISTERS:         /* 0x03 */
    case MBT_READ_INPUT_REGISTERS:           /* 0x04 */
      if (inst->uiReadQty > MAX_REGISTER) //same value as Holding register
         { inst->uiStatus = mbtERR_MAX_NBR_REGISTER; inst->bRecvOK = FALSE; goto END; }
      break;
    case MBT_WRITE_SINGLE_COIL:              /* 0x05 */
    case MBT_WRITE_MULTIPLE_COILS:           /* 0x0F */
     if (inst->uiWriteQty > MAX_COILS)
         { inst->uiStatus = mbtERR_MAX_NBR_COILS; inst->bRecvOK = FALSE; goto END; }
      break;
    case MBT_WRITE_SINGLE_REGISTER:          /* 0x06 */
    case MBT_WRITE_MULTIPLE_REGISTERS:       /* 0x10 */
      if (inst->uiWriteQty > MAX_REGISTER)
        { inst->uiStatus = mbtERR_MAX_NBR_REGISTER; inst->bRecvOK = FALSE; goto END; }
      break;
    case MBT_READ_WRITE_MULTIPLE_REGISTER:  /* 0x17 */
      if (    (inst->uiWriteQty > MAX_REGISTER)
           || (inst->uiReadQty > MAX_REGISTER))
        { inst->uiStatus = mbtERR_MAX_NBR_REGISTER; inst->bRecvOK = FALSE; goto END; }
      break;
    default:
      { inst->uiStatus = mbtERR_ILLEGAL_FUNCTION; goto END; }
    }

    switch(inst->usiFCode)
    {
    case MBT_READ_COILS:                     /* 0x01 */
    case MBT_READ_DISCRETE_INPUTS:           /* 0x02 */
    case MBT_READ_HOLDING_REGISTERS:         /* 0x03 */
    case MBT_READ_INPUT_REGISTERS:           /* 0x04 */
      if(inst->puiReadVal == NULL)
        { inst->uiStatus = mbtERR_DATA_ADDRESS; goto END; }
      mbm->pData->actParam[0].puiReadVal = (UDINT) inst->puiReadVal;
      break;
    case MBT_WRITE_SINGLE_COIL:              /* 0x05 */
    case MBT_WRITE_MULTIPLE_COILS:           /* 0x0F */
    case MBT_WRITE_SINGLE_REGISTER:          /* 0x06 */
    case MBT_WRITE_MULTIPLE_REGISTERS:       /* 0x10 */
      if( inst->puiWriteVal == NULL)
        { inst->uiStatus = mbtERR_DATA_ADDRESS; goto END; }
      mbm->pData->actParam[0].puiWriteVal = (UDINT) inst->puiWriteVal;
      break;
    case MBT_READ_WRITE_MULTIPLE_REGISTER:  /* 0x17 */
      if(    (inst->puiWriteVal == NULL)
          || (inst->puiReadVal == NULL))
        { inst->uiStatus = mbtERR_DATA_ADDRESS; goto END; }
      mbm->pData->actParam[0].puiReadVal  = (UDINT) inst->puiReadVal;
      mbm->pData->actParam[0].puiWriteVal = (UDINT) inst->puiWriteVal;
      break;
    default:
      { inst->uiStatus = mbtERR_ILLEGAL_FUNCTION; goto END; }
    }

    inst->bRecvOK = mbm->bRecvOK;
    inst->uiStatus = ERR_OK;
  }
END: ; /* do nothing */
  /*=========================================================================*/
} /* fMBTMRW */

/*****************************************************************************
 * END OF CODE
 *****************************************************************************/
/*
  Local Variables:
  c-file-style: bsd
  c-basic-offset: 2
  comment-column: 45
  End:
*/
```
